// TwinCAT 3 PLC project RS485HausBus
// ProgramVersion: 3.1.4024.0
// libraries:
//   Tc2_SerialCom, * (Beckhoff Automation GmbH)
//   Tc2_Standard, * (Beckhoff Automation GmbH)
//   Tc2_System, * (Beckhoff Automation GmbH)
//   Tc3_Module, * (Beckhoff Automation GmbH)
// project tree:
//   DUTs/BusTaster/ ST_BusTaster6F_Cnt.TcDUT, ST_BusTaster6F_Input.TcDUT (not stored), ST_BusTaster6F_Output.TcDUT (not stored)
//   DUTs/RelaisModul/ ST_BusRelais16F_Cnt.TcDUT (not stored), ST_BusRelais16F_Input.TcDUT (not stored), ST_BusRelais16F_Output.TcDUT (not stored)
//   DUTs/Service/ ST_FiFoMaster_State.TcDUT (not stored), ST_RS485Startup_State.TcDUT
//   / GlobalTextList.TcGTLO, PlcTask.TcTTO, Visualisierungsmanager.TcVMO (not stored)
//   GVLs/ GVL.TcGVL, GVL_Constant.TcGVL, GVL_HausBus_Parameter.TcGVL (not stored), GVL_RS485FiFoSend.TcGVL, GVL_ServiceVisu.TcGVL
//   POUs/ RS485_COM_PRG.TcPOU
//   POUs/RS485_Hausbus_FB/BusTaster/ fb_StringConvTB6F.TcPOU, fb_TasterBus6F.TcPOU
//   POUs/RS485_Hausbus_FB/Events/ fb_BusBrsEvent.TcPOU, fb_BusPingEvent.TcPOU, fb_BusRhdEvent.TcPOU, fb_BusTasterEvent.TcPOU, fb_BusTempEvent.TcPOU
//   POUs/RS485_Hausbus_FB/RelaisModul/ fb_RelaisBus16F.TcPOU, fb_StringConvRB16F.TcPOU
//   POUs/RS485_Hausbus_FB/RS485 COM/FB/ fb_FilterArray.TcPOU
//   POUs/RS485_Hausbus_FB/RS485 COM/ fb_RS485ComCheck.TcPOU
//   POUs/RS485_Hausbus_FB/RS485 COM/RS485_Master/ fb_RS485FiFoMaster.TcPOU, fb_RS485Startup.TcPOU
//   VISUs/HausBus_RS485/ BusRelais16F_Frame.TcVIS, BusRS485Master_Frame.TcVIS, BusTatster6F_Frame.TcVIS, RS485HB_ServiceVISU.TcVIS

CONFIGURATION RS485HausBus
    RESOURCE PLC ON TwinCAT3
        TASK PlcTask(INTERVAL := T#1ms, PRIORITY := 20);
        PROGRAM RS485_COM_PRG WITH PlcTask : RS485_COM_PRG;
    END_RESOURCE
END_CONFIGURATION

// ---- DUTs/BusTaster/ST_BusTaster6F_Cnt.TcDUT
TYPE ST_BusTaster6F_Cnt :
STRUCT
	dwCntButtons    :ARRAY[1..6] OF DWORD;
END_STRUCT
END_TYPE

// ---- DUTs/Service/ST_RS485Startup_State.TcDUT
TYPE ST_RS485Startup_State :
STRUCT
	bBusOk					:BOOL;
	bStartupError			:BOOL;
	sStartupState			:STRING;
	bStartupDone			:BOOL;
END_STRUCT
END_TYPE

// ---- GVLs/GVL.TcGVL
{attribute 'Tc2GvlVarNames'}
VAR_GLOBAL

    KL6041In    					AT %I* : KL6inData22B; // Eingangsdaten von der Klemme
    KL6041Out 						AT %Q* : KL6outData22B; // Ausgangsdaten zur Klemme
	
	uiEtherCATStateBK1120_RS485COM	AT %I* : UINT;			// EtherCAT Status 
	uiKBusStateBK1120_RS485COM		AT %I* : UINT;			// Buskoppler Status
	
END_VAR

// ---- GVLs/GVL_Constant.TcGVL
{attribute 'Tc2GvlVarNames'}
VAR_GLOBAL CONSTANT
	cMaxBusTaster	:INT :=10;			// Anzahl der Bus Taster 
	cMaxBusRelais	:INT :=1;			// Anzahl der Bus Relais 
	cMaxRS485CMDFiFo	:INT := 15;		// Anzahl der Zeilen im FiFo Buffer (Achtung jder Bus Teilnehmer Benötigt eine Zeile! also immer cMaxBusTaster +cMaxBusRelais +etc.)  
END_VAR

// ---- GVLs/GVL_RS485FiFoSend.TcGVL
{attribute 'qualified_only'}
VAR_GLOBAL
	bSendDoneFiFo	:ARRAY[1..cMaxRS485CMDFiFo] OF BOOL;			(* Rückmeldung Aus dem FiFo Master Baustein, dass der Sendevorgang abgeschlossen ist *)
	sSendFiFo		:ARRAY[1..cMaxRS485CMDFiFo] OF STRING(255);		(* Zeile für den FiFo Master Baustein, von jedem einzelnen Busteilnehmer *)
END_VAR

// ---- GVLs/GVL_ServiceVisu.TcGVL
{attribute 'qualified_only'}
VAR_GLOBAL
	iDeviceTasterVisu			:INT := 1;
	iDeviceRelaisVisu			:INT := cMaxBusTaster+1;
	
	bTasterServiceAktiv			:ARRAY[1..cMaxBusTaster] OF BOOL;
	bRelaisServiceAktiv			:ARRAY[cMaxBusTaster+1..cMaxBusTaster+cMaxBusRelais+1] OF BOOL;
	stTasterService				:ARRAY[1..cMaxBusTaster] OF ST_BusTaster6F_Input;
	stRelaisService				:ARRAY[cMaxBusTaster+1..cMaxBusTaster+cMaxBusRelais+1] OF ST_BusRelais16F_Input;
	
END_VAR

// ---- POUs/RS485_COM_PRG.TcPOU
(*======================================================================================================================================*)
(*RS485_COM_PRG: Beispielhaftes Programm zum Steuern von HAus-Bus.de Komponenten über RS485 mit TwinCAT
					Achtung dieser POU muss als 1ms Task Aufgerufen werden um Ordnungsgemäß zu laufen *)
(*
Date          	| Version    	| created under        	| Author          	| Remark *)
(*====================================================================================================================================================*)
(*15/05/2025   	| 1.00      		| TC3		  		| N.Kersting       | first release *)
(*====================================================================================================================================================*)

PROGRAM RS485_COM_PRG
VAR  
    fbTaster 					:ARRAY[1..cMaxBusTaster] OF fb_TasterBus6F;	
	fbRelais					:ARRAY[cMaxBusTaster+1..cMaxBusRelais+cMaxBusTaster+1] OF fb_RelaisBus16F;
    i,h,j						:INT;
	
	fbRS485Startup				:fb_RS485Startup;		(* Startup Parametrierung der Klemme/ RS485 Bus *)
	fbRS485SendCmdFiFo			:fb_RS485FiFoMaster;	(* Sende und Empfangs FiFo für RS485 *)
	fbLineControl 				:SerialLineControl;		(* Hält die Serielle Kommunikation Aufrecht *)
	
	fComBufferReset				:ClearComBuffer;		(* Löschen des SPS Internen Bufferinhalts *)
	
	rxBuffer 					:ComBuffer;				(* COM Buffer Empfangen *)
    txBuffer 					:ComBuffer;				(* COM Buffer Senden *)
	
	
	
END_VAR

(* IDs Setzen *)
ac00_HausBusIdRS485COM();
(* RS485 Klemmen Config *)
ac01_StartupRS485COM();

ACTION ac00_HausBusIdRS485COM:
(* Initialisierung der Gerätenamen *)
(* Achtung nur Beispiele *)
fbTaster[1].I_stInput.sName := 		'Wohnzimmer';		(* Name, wie der Teilnehmer heißt / Bezeichnung *)
fbTaster[1].I_stInput.diID := 		5256;				(* Haus-Bus ID, welche auf dem Aufkleber steht  *)
		
fbTaster[2].I_stInput.sName := 		'Test1';
fbTaster[2].I_stInput.diID := 		5269;

fbTaster[3].I_stInput.sName := 		'Test2';
fbTaster[3].I_stInput.diID := 		2222;

fbTaster[4].I_stInput.sName := 		'Test3';
fbTaster[4].I_stInput.diID := 		3333;

fbTaster[5].I_stInput.sName := 		'Test4';
fbTaster[5].I_stInput.diID := 		4444;

fbTaster[6].I_stInput.sName := 		'Test5';
fbTaster[6].I_stInput.diID := 		5555;

fbTaster[7].I_stInput.sName := 		'Test6';
fbTaster[7].I_stInput.diID := 		6666;

fbTaster[8].I_stInput.sName := 		'Test7';
fbTaster[8].I_stInput.diID := 		7777;

fbTaster[9].I_stInput.sName := 		'Test8';
fbTaster[9].I_stInput.diID := 		8888;

fbTaster[10].I_stInput.sName := 	'Test9';
fbTaster[10].I_stInput.diID := 		9999;

fbRelais[11].I_stInput.sName := 	'Jalousie 1';
fbRelais[11].I_stInput.diID :=		5614;
END_ACTION

ACTION ac01_StartupRS485COM:

(* Klemmen Startup, inkl Klemmenkonfiguration usw. *)
fbRS485Startup(
	I_bExecute:= 		TRUE, 
	I_bBusOK:= 			uiEtherCATStateBK1120_RS485COM = 8
						AND uiKBusStateBK1120_RS485COM = 0, 
	I_tStartupVerz:= 	T#5S, 
	IQ_InData:= 		KL6041In, 
	IQ_OutData:= 		KL6041Out, 
	Q_sState=> , 
	Q_bStartupDone=> , 
	Q_bError=> );

(* Aktivierung der Linecontrole erst wenn Startup erfolgt *)	
IF fbRS485Startup.Q_bStartupDone
THEN
	fbLineControl(
		Mode := 		ComSerialLineMode_t.SERIALLINEMODE_KL6_22B_STANDARD,
		pComIn := 		ADR(KL6041In),
		pComOut := 		ADR(KL6041Out),
		SizeComIn := 	UINT_TO_INT(SIZEOF(KL6041In)),
		RxBuffer := 	rxBuffer,
		TxBuffer := 	txBuffer );
				
	(* Relais *)
	ac10_HausBusRelaisRS485COM();
	(* Taster *)
	ac10_HausBusTasterRS485COM();
	
	(* Senden FiFo *)
	fbRS485SendCmdFiFo(
		I_sSendCmdFiFo:= 		GVL_RS485FiFoSend.sSendFiFo, 
		I_bExecute:= 			TRUE, 
		I_bBusBelastungstest := ,
		I_bReset:= , 
		I_pTxBuffer:= 			ADR(txBuffer), 
		I_pRxBuffer:= 			ADR(rxBuffer), 
		Q_lrBusAuslastung=>		,
		Q_bBusy=> , 
		Q_bDone=> , 
		Q_bError=> , 
		Q_sState=> );
	
ELSE
	(* Com Buffer zum Resetten *)
	fComBufferReset(Buffer:= rxBuffer);
	fComBufferReset(Buffer:= txBuffer);
END_IF
END_ACTION

ACTION ac10_HausBusRelaisRS485COM:
(* BusRelais Aufrufe *)
FOR h := cMaxBusTaster +1 TO cMaxBusRelais+cMaxBusTaster+1 BY 1 DO (*cMaxBusTaster+1..cMaxBusRelais+cMaxBusTaster+1*)
		
	IF GVL_ServiceVisu.bRelaisServiceAktiv[h]
	THEN
		fbRelais[h].I_stInput.bOut := GVL_ServiceVisu.stRelaisService[h].bOut;
		fbRelais[h].I_stInput.bReset := GVL_ServiceVisu.stRelaisService[h].bReset;
	END_IF
	
	GVL_ServiceVisu.stRelaisService[h].sName :=	fbRelais[h].I_stInput.sName;
	GVL_ServiceVisu.stRelaisService[h].diID :=	fbRelais[h].I_stInput.diID;
	
	fbRelais[h].I_stInput.bExecute := TRUE;
	fbRelais[h](
		I_FifoID :=			h,
		I_bPingStart:= 		TRUE,	(* Direkt Starten *)
		I_StringReceived:=	fbRS485SendCmdFiFo.Q_sReceiveString);
		
	(* Sendebefehle an FiFo Übergeben *)
	GVL_RS485FiFoSend.sSendFiFo[h] :=	fbRelais[h].Q_sFiFoSend;	
END_FOR
END_ACTION

ACTION ac10_HausBusTasterRS485COM:
(* Bustaster Aufrufe *)
FOR i := 1 TO cMaxBusTaster BY 1 DO
			
	IF GVL_ServiceVisu.bTasterServiceAktiv[i]
	THEN
		fbTaster[i].I_stInput.iLED := GVL_ServiceVisu.stTasterService[i].iLED;
		fbTaster[i].I_stInput.iLEDBg := GVL_ServiceVisu.stTasterService[i].iLEDBg;
		fbTaster[i].I_stInput.iLEDExt := GVL_ServiceVisu.stTasterService[i].iLEDExt;
		fbTaster[i].I_stInput.bReset := GVL_ServiceVisu.stTasterService[i].bReset;
	END_IF
	
	GVL_ServiceVisu.stTasterService[i].sName :=	fbTaster[i].I_stInput.sName;
	GVL_ServiceVisu.stTasterService[i].diID :=	fbTaster[i].I_stInput.diID;
	
	fbTaster[i].I_stInput.bExecute := TRUE;
	fbTaster[i](
		I_FifoID :=			i,
		I_bPingStart:= 		TRUE , 	(* Taster Verzögert Pingen, damit weniger Busauslastung entsteht *)
		I_StringReceived:=	fbRS485SendCmdFiFo.Q_sReceiveString);
		
	(* Sendebefehle an FiFo Übergeben *)
	GVL_RS485FiFoSend.sSendFiFo[i] :=	fbTaster[i].Q_sFiFoSend;
END_FOR
END_ACTION

END_PROGRAM

// ---- POUs/RS485_Hausbus_FB/BusTaster/fb_TasterBus6F.TcPOU
(*======================================================================================================================================*)
(*FB_TasterBusSimple:	Einfache RS485 Kommunikation für Haus-bus.de Komponenten zum testen 	
						Achtung: Bei dem 6 Fach Taster ist zu Beachten, dass es nur 4 Externe EA/s gibt also 4 LEDs und 4 Taster *)
(*
Date          	| Version    	| created under        	| Author          	| Remark *)
(*====================================================================================================================================================*)
(*29/04/2025   	| 1.00      		| TC3		  		| N.Kersting       | first release *)
(*02/05/2025   	| 1.01      		| TC3		  		| N.Kersting       | Events für die Buttons werden erfolgreich verarbeitet *)
(*02/05/2025   	| 1.02      		| TC3		  		| N.Kersting       | Events für Temp, Helligkeit, Fuehctigkeit erfolgreich Implementier *)
(*02/05/2025   	| 1.03      		| TC3		  		| N.Kersting       | Set Schrittkette für Reset und LED Helligkeit erfolgreich Implementier*)
(*02/05/2025   	| 1.04      		| TC3		  		| N.Kersting       | In und Out Strukturen Implementiert und Startup nach Reset *)
(*02/05/2025   	| 1.05      		| TC3		  		| N.Kersting       | Pingabgfrage*)
(*02/05/2025   	| 1.06      		| TC3		  		| N.Kersting       | Reset Startup Implementiert*)
(*03/05/2025   	| 1.07      		| TC3		  		| N.Kersting       | Ping wird nun bei PLC Reset auch gestaret und Execute wird richtig verwendet*)
(*04/05/2025   	| 1.08      		| TC3		  		| N.Kersting       | Hintergrundbeleuchtung und Zähler für die Tatser Implementiert *)
(*04/05/2025   	| 1.09      		| TC3		  		| N.Kersting       | Neuen Baustein zum Einheitlichen versenden von Telegrammen Implementiert *)
(*05/05/2025   	| 2.00      		| TC3		  		| N.Kersting       | Komplett neuen Baustein, mit Externer Receive Auswertung und neuem Ping Baustein *)
(*06/05/2025   	| 2.01      		| TC3		  		| N.Kersting       | Externe LEDs Implementiert *)
(*07/05/2025   	| 2.02      		| TC3		  		| N.Kersting       | Im Startup wird nun auf die Device ID geachtet *)
(*08/05/2025   	| 2.03      		| TC3		  		| N.Kersting       | Externe LEDs sind nun Umschaltbar/ LEDs oder normaler Ausgang (Betriefft die Hintergrundbeleuchtung) -> Weniger Busauslastung *)
(*09/05/2025   	| 2.04      		| TC3		  		| N.Kersting       | Ping Versuche Implementiert mit Globalen Parametern *)
(*09/05/2025   	| 2.05      		| TC3		  		| N.Kersting       | Ping für Taster nun Auch automatisch durch Empfang von sämtlichen Telegrammen*)
(*09/05/2025   	| 2.06      		| TC3		  		| N.Kersting       | Bugfix im Startup Angepasst! nur noch Hintergrundbeleuchtung setzen! *)
(*10/05/2025   	| 3.00      		| TC3		  		| N.Kersting       | Umstellung auf Externe FiFo Sendebaustein *)
(*13/05/2025   	| 3.01      		| TC3		  		| N.Kersting       | Viele Bugs gefixt, bei Änderung der Ausgängen wird nun eine Anforderung gesetzt  *)
(*13/05/2025   	| 3.02      		| TC3		  		| N.Kersting       | Test für Github *)
(*====================================================================================================================================================*)
FUNCTION_BLOCK fb_TasterBus6F
VAR_INPUT
	I_FifoID			:INT;
	I_bPingStart		:BOOL;						(* Ping Done vom Vorheriegen*)
	I_stInput			:ST_BusTaster6F_Input;
	I_StringReceived	:STRING(255);
END_VAR
VAR_OUTPUT
	Q_sFiFoSend			:STRING(255);
   	Q_stOutput			:ST_BusTaster6F_Output;
	Q_stCnt				:ST_BusTaster6F_Cnt;
END_VAR
VAR
(*----------------------------------------------*)
(* Interne Parameter*)
(*----------------------------------------------*)		
	bSetExecute			:BOOL := TRUE;				(* Aktiviert die Schrittketten, welche Telegramme versenden *)
	bCheckPing			:BOOL := TRUE;				(* Ping Checken Schrittkette Aktivieren *)
	sStartZeichen		:BYTE := 16#FD;				(* Startzeichen Präfix *)
	sEndZeichen			:BYTE := 16#FE;				(* Endzeichen Suffix *)
	iAnzResetSend		:INT := 2;					(* Anzahl der Sendeversuche bei Reset *)
	tPingTimer			:TIME:= T#5S;				(* Zeit, bis wiederholend der Ping versendet wird *)
	tReceiveTimeout		:TIME:= T#2S;				(* Zeit, bis die Event Schrittkette für das Empfangen Automatisch neu Startet*)
	tStartupLEDOn		:TIME:= T#4S;				(* Zeit, wie Lange die LEDS beim Startup kurz eingeschaltet werden *)
	tResetTimeout		:TIME:= T#8S;				(* Zeit, bis bei einem Reset es zu einem Fehler kommt, wenn kein Ping empfangen wird *)
	tResetReboot		:TIME:= T#10S;				(* Zeit, die nach einem Reset Abgewaretet wird damit das Gerät neustarten kann*)
	tResetStartup		:TIME:= T#5S;				(* Zeit, die nach einem Reset Abgewaretet wird bis ein Startup ausgeführt wird nach dem erhalt des Pings vom Gerät*)
	tStartupAfterReset	:TIME := T#5S;				(* Zeit, wann das Startup Zurückgesetzt wird, wenn der Ping verloren wird *)
(*----------------------------------------------*)
(* Strings *)
(*----------------------------------------------*)			
	sSendString			:STRING(255);
	sFiFoSend			:STRING(255);
	sReceived			:STRING(255);
	sLastSendString		:STRING(255);
	sStateReset			:STRING;
(*----------------------------------------------*)
(* Funktionsbausteine *)
(*----------------------------------------------*)
	fbBusTasterEvent	:ARRAY[1..6] OF fb_BusTasterEvent;		(* Interne 6 Taster Abfragen *)
	fbBusTasterEventExt	:ARRAY[1..6] OF fb_BusTasterEvent;		(* Externe 6 Eingänge Abfragen *)
	fbBusTempEvent		:fb_BusTempEvent;
	fbBusBrsEvent		:fb_BusBrsEvent;
	fbBusRhdEvent		:fb_BusRhdEvent;
	fbStringConvTB6F	:fb_StringConvTB6F;
	fbRS485ComCheck		:fb_RS485ComCheck;
(*----------------------------------------------*)
(* Indexe *)
(*----------------------------------------------*)	
	iDeviceStartup		:INT :=0;	(* Startup Schrittkette *)
	sDeviceStartup		:STRING;
    iState     			:INT := 0;
	iStepSet			:INT;
	i,h,j,l,e			:INT;
	idxLED				:INT;
	idxBtn				:INT := 1;
	
	iDimmMem			:ARRAY[1..6] OF INT;
	iDimmMemExt			:ARRAY[1..6] OF INT;
	iDimmBGAnf			:INT;
	iDimmAnf			:ARRAY[1..6] OF INT;
	iDimmAnfExt			:ARRAY[1..6] OF INT;
	
	iDimmBgMem			:INT;
	cntChangesDimm		:INT;
	cntChangesDimmExt	:INT;
	icntResetSend		:INT;
	iMaxPingTry			:INT := 5;
(*----------------------------------------------*)
(* Timer/Trigger *)
(*----------------------------------------------*)		
	r_trigStartupAfterReset	:r_trig;
	r_TrigReset				:r_trig;		
	r_TrigCountBtn			:ARRAY[1..6] OF r_trig;
	
	tonStartupAfterReset	:ton;
	tonReceiveTimeout		:ton;
	tonResetTimeout			:ton;
	tonResetDone			:ton;
	tonStepStartup			:ton;
(*----------------------------------------------*)
(* Status *)
(*----------------------------------------------*)			
	bPingOK					:BOOL;
	bErrorEvent				:BOOL;
	bErrorPing				:BOOL;
	bErrorSet				:BOOL;
	bErrorReset				:BOOL;
	bResetBusy				:BOOL;
	bResetDone				:BOOL;
	bResetAutoStart			:BOOL;
	bStartupStart			:BOOL;
	bStartupDone			:BOOL;	
	bMemExt					:BOOL;
	bStartUpCheckPing		:BOOL;
	bActivateSend			:BOOL;
	bReadyToPing			:BOOL;
	bSendeAnforderung		:BOOL;
	bSendeAnforderungExt	:BOOL;
	bSendeAnforderungBG		:BOOL;
	
END_VAR

(*============================================================================================*)
(* Parameter *)
tPingTimer :=		GVL_HausBus_Parameter.cTimePingTimeTaster;
tReceiveTimeout :=	GVL_HausBus_Parameter.cTimeReceiveTimeoutTaster;
bCheckPing :=		GVL_HausBus_Parameter.bUseTasterPing;
iMaxPingTry :=		GVL_HausBus_Parameter.cMaxPingTry;

(*============================================================================================*)
(* Startup Zurücksetzen Reset *)
r_TrigReset(CLK := I_stInput.bReset);

(* Startup Zurücksetzen bei Busverlust *)
tonStartupAfterReset(
	IN := NOT bPingOK
			AND bCheckPing,
	PT:= tStartupAfterReset);

r_trigStartupAfterReset
	(CLK := tonStartupAfterReset.Q);
	
IF NOT I_stInput.bExecute
	OR r_TrigReset.Q
	OR r_trigStartupAfterReset.Q
THEN
	iDeviceStartup := 0;
END_IF

(*============================================================================================*)
(* Ping Dauerhaft Senden*)
ac02_Ping();
	
(*============================================================================================*)
(* Startup Schrittkette *)
CASE iDeviceStartup OF
(*============================================================================================*)
0: 	sDeviceStartup := 'INIT';
	bResetDone := FALSE;
	bStartupDone := FALSE;
	bStartupStart := FALSE;
	bResetAutoStart := FALSE;
	bStartUpCheckPing := FALSE;
	bActivateSend := FALSE;
	bReadyToPing := TRUE;
	sFiFoSend := ''; 
	iStepSet := 0;
	
	IF 	I_stInput.bExecute
	THEN
		iDeviceStartup := iDeviceStartup+1;
	END_IF
(*============================================================================================*)
1: 	sDeviceStartup := 'Device ID Prüfen';
	
	IF  I_stInput.diID <> 0
	THEN
		iDeviceStartup := iDeviceStartup+1;
	ELSE
		sDeviceStartup := 'ERROR- Device ID Prüfen';
	END_IF
(*============================================================================================*)
2: 	sDeviceStartup := 'Verbindung Prüfen';
	bStartUpCheckPing := TRUE;
	bActivateSend := TRUE;	(* Senden Aktivieren *)
	
	sDeviceStartup := CONCAT(sDeviceStartup,fbRS485ComCheck.Q_sState);
	
	IF fbRS485ComCheck.Q_bComOk
		OR NOT bCheckPing
	THEN
		iDeviceStartup := iDeviceStartup+1;
	END_IF

(*============================================================================================*)
3: 	sDeviceStartup := 'Reset Ausführen';	
	bActivateSend := TRUE;	(* Senden Aktivieren *)
	
	(*	RESET Device *)
	ac01_SetReset();
	bResetAutoStart := TRUE;
	
	sDeviceStartup :=	CONCAT(sDeviceStartup,sStateReset);
	
	IF bResetDone
	THEN
		iStepSet := 0;
		iDeviceStartup := iDeviceStartup+1;
	END_IF

(*============================================================================================*)
4: 	sDeviceStartup := 'Startup Ausführen';
		
	(* LED Setzen *)
	ac01_SetLED();
	
	bStartupStart := TRUE;
	
	IF bStartupDone 
	THEN
		bStartupStart := FALSE;
		iDeviceStartup := 999;
	END_IF

(*============================================================================================*)
999: 
	(*bReadyToPing := NOT fbRS485SendCmd.Q_bBusy;*)
	
	(* LED Setzen *)
	ac01_SetLED();
	
	(* Events Auslesen *)
	ac00_Event();
	
	(* Zähler *)
	ac10_Counter();
	
	sDeviceStartup := 'Startup Ausgeführt- Gerät im OP';
	
END_CASE

(*============================================================================================*)
(* Sendebaustein *)
IF bActivateSend
THEN
	IF fbRS485ComCheck.Q_sSend <>''
	THEN
		Q_sFiFoSend :=	fbRS485ComCheck.Q_sSend;
	ELSE
		Q_sFiFoSend :=	sFiFoSend;
	END_IF
END_IF

(*============================================================================================*)	
(* Zähler *)
ac10_Counter();
	
(*============================================================================================*)
(* Outputs *)
Q_stOutput.bCOM :=		bPingOK;

Q_stOutput.bError := 	bErrorEvent
						OR bErrorPing
						OR bErrorSet
						OR (NOT bPingOK
						AND bCheckPing);
						
Q_stOutput.bStartupDone	:=	bStartupDone;

Q_stOutput.sState :=	CONCAT(I_stInput.sName,'| ');
Q_stOutput.sState :=	CONCAT(Q_stOutput.sState, sDeviceStartup);

ACTION ac00_Event:
(*============================================================================================*)
(*	EVENT Schrittkette *)
(*============================================================================================*)
sReceived := I_StringReceived;
	
FOR i := 1 TO 6 BY 1 DO 
	fbBusTasterEvent[i](
		I_sID:= 				DINT_TO_STRING(I_stInput.diID), 
		I_sInstID:= 			INT_TO_STRING(i+16), 
		I_sReceivedString:= 	sReceived, 
		Q_bOut=> 				Q_stOutput.bButtons[i]);
	
	fbBusTasterEventExt[i](
		I_sID:= 				DINT_TO_STRING(I_stInput.diID), 
		I_sInstID:= 			INT_TO_STRING(i+32), 
		I_sReceivedString:= 	sReceived, 
		Q_bOut=> 				Q_stOutput.bButtonsExt[i]);
		
	fbBusTempEvent(
		I_sID:= 				DINT_TO_STRING(I_stInput.diID), 
		I_sInstID:= 			'1', 
		I_sReceivedString:= 	sReceived, 
		Q_lrTemp=> 				Q_stOutput.lrTemp);
		
	fbBusBrsEvent(
		I_sID:= 				DINT_TO_STRING(I_stInput.diID), 
		I_sInstID:= 			'1', 
		I_sReceivedString:= 	sReceived, 
		Q_lrBrs=> 				Q_stOutput.lrBrs);
		
	fbBusRhdEvent(
		I_sID:= 				DINT_TO_STRING(I_stInput.diID), 
		I_sInstID:= 			'1', 
		I_sReceivedString:= 	sReceived, 
		Q_lrRhd=> 				Q_stOutput.lrRhd);
END_FOR
END_ACTION

ACTION ac01_SetLED:
(*============================================================================================*)
(*	LED Helligkeit Setzen/ Startup Schrittkette *)
(*============================================================================================*)

(* Einfaches Setzen der LED Helligkeiten (0-100 Prozent *)
(* Neu, es werden alle LEDs zu einem String zusammengefügt und Gleichzeitig gesetzt *)
tonStepStartup(
	PT:= tStartupLEDOn);
	
cntchangesDimm := 0;
cntChangesDimmExt :=0;
	
FOR l := 1 TO 6 BY 1 DO
	IF iDimmMem[l] <> I_stInput.iLED[l]
	THEN
		cntChangesDimm := cntChangesDimm +1;
	END_IF

	IF  iDimmMemExt[l]<> I_stInput.iLEDExt[l]
	THEN
		cntChangesDimmExt := cntChangesDimmExt +1;
	END_IF
END_FOR

CASE iStepSet OF
(*============================================================================================*)
0:	(* INIT und warten auf Change *)				
	tonStepStartup.IN := FALSE;
	sFiFoSend := ''; 
	
	(* Änderungs- Anforderungen Prüfen*)
	FOR e := 1 TO 6 BY 1 DO
		IF cntChangesDimm<>0
		THEN
			(* Helligkeitanforderung Interne LEDs speichern *)
			bSendeAnforderung := TRUE;
			iDimmAnf[e] 	:= I_stInput.iLED[e];
		END_IF
		
		IF cntChangesDimmExt <> 0
		THEN
			(* Helligkeitanforderung Externe LEDs speichern *)
			bSendeAnforderungExt := TRUE;
			iDimmAnfExt[e] 	:= I_stInput.iLEDExt[e];
		END_IF
		
		IF I_stInput.iLEDBg <>iDimmBgMem
		THEN
			(* Helligkeitsanforderung Hintergrundbeleuchtung *)
			bSendeAnforderungBG := TRUE;
			iDimmBGAnf		:= I_stInput.iLEDBg;
		END_IF
	END_FOR
	
	(* Reagieren auf Anforderungen *)
	IF ((bSendeAnforderung
		OR bSendeAnforderungExt
		OR bSendeAnforderungBG)
		AND bSetExecute)
		AND fbRS485ComCheck.Q_sSend =''
		AND NOT bStartupStart
	THEN
		(* Helligkeitsvorgaben speichern in Mem Arrays *)
		FOR h := 1 TO 6 BY 1 DO
			iDimmMem[h] := I_stInput.iLED[h];
			iDimmMemExt[h] := I_stInput.iLEDExt[h];
			iDimmBgMem := I_stInput.iLEDBg;
		END_FOR
		
		iStepSet := 10;
	ELSIF
		bStartupStart
	THEN
		iStepSet := 100;	(* Startup *)
	END_IF
	
(*============================================================================================*)
10:	(* Prüfen welche Anforderung ausgeführt werden soll *)	
	IF	bSendeAnforderungBG
		AND NOT bSendeAnforderung
		AND NOT bSendeAnforderungExt 
	THEN
		iStepSet := 22;(* Direkt nur die Hintergrund Helligkeit setzen *)
	ELSE
		(* Nur Interne LEDs Schreiben *)
		IF bSendeAnforderung
			AND NOT bSendeAnforderungExt
			AND NOT bSendeAnforderungBG
		THEN
			fbStringConvTB6F(
				I_bSetBackground :=	FALSE,
				I_bReset :=			FALSE,
				I_bExtLED :=		FALSE,
				I_bHasExtLED :=		I_stInput.bExtOutLED,
				I_diID:= 			I_stInput.diID, 
				I_iLED:= 			iDimmAnf, 
				I_iLEDExt:=			iDimmAnfExt,
				I_iLEDBg:= 			iDimmBGAnf,		 
				I_sStartZeichen:= 	sStartZeichen, 
				I_sEndZeichen:= 	sEndZeichen, 
				Q_sConvString=> 	sSendString);
				
			(* Senden an FiFo*)
			IF GVL_RS485FiFoSend.bSendDoneFiFo[I_FifoID]
			THEN
				sFiFoSend :=	sSendString;
			END_IF
			IF NOT GVL_RS485FiFoSend.bSendDoneFiFo[I_FifoID]
			THEN
				bSendeAnforderung := FALSE;
				sLastSendString :=	sFiFoSend;
				iStepSet := 20;
			END_IF
		ELSIF
			(* Nur Externe LEDs Schreiben *)	
			bSendeAnforderungExt
			AND NOT bSendeAnforderung
			AND NOT bSendeAnforderungBG
		THEN
			fbStringConvTB6F(
				I_bSetBackground :=	FALSE,
				I_bReset :=			FALSE,
				I_bExtLED :=		TRUE,
				I_bHasExtLED :=		I_stInput.bExtOutLED,
				I_diID:= 			I_stInput.diID, 
				I_iLED:= 			iDimmAnf, 
				I_iLEDExt:=			iDimmAnfExt,
				I_iLEDBg:= 			iDimmBGAnf,				 
				I_sStartZeichen:= 	sStartZeichen, 
				I_sEndZeichen:= 	sEndZeichen, 
				Q_sConvString=> 	sSendString);
			
			(* Senden an FiFo*)
			IF GVL_RS485FiFoSend.bSendDoneFiFo[I_FifoID]
			THEN
				sFiFoSend :=	sSendString;
			END_IF
			IF NOT GVL_RS485FiFoSend.bSendDoneFiFo[I_FifoID]
			THEN
				bSendeAnforderungExt := FALSE;
				sLastSendString :=	sFiFoSend;
				iStepSet := 20;
			END_IF
		ELSE
			(* Externe und Interne LEDs Schreiben *)
			bMemExt := TRUE; (* Speichern, damit anschließend noch die Externen LEDs gesetzt werden *)
			
			fbStringConvTB6F(
				I_bSetBackground :=	FALSE,
				I_bReset :=			FALSE,
				I_bExtLED :=		FALSE,
				I_bHasExtLED :=		I_stInput.bExtOutLED,
				I_diID:= 			I_stInput.diID, 
				I_iLED:= 			iDimmAnf, 
				I_iLEDExt:=			iDimmAnfExt,
				I_iLEDBg:= 			iDimmBGAnf,			 
				I_sStartZeichen:= 	sStartZeichen, 
				I_sEndZeichen:= 	sEndZeichen, 
				Q_sConvString=> 	sSendString);
			
			(* Senden an FiFo*)
			IF GVL_RS485FiFoSend.bSendDoneFiFo[I_FifoID]
			THEN
				sFiFoSend :=	sSendString;
			END_IF
			IF NOT GVL_RS485FiFoSend.bSendDoneFiFo[I_FifoID]
			THEN
				bSendeAnforderung := FALSE;
				bSendeAnforderungExt := FALSE;
				sLastSendString :=	sFiFoSend;
				iStepSet := 20;
			END_IF
		END_IF
	END_IF
(*============================================================================================*)	
20:	(* Warten bis nicht Busy *)	
	
	IF GVL_RS485FiFoSend.bSendDoneFiFo[I_FifoID]
	THEN
		sFiFoSend := ''; 
		IF NOT bMemExt
		THEN
			IF bSendeAnforderungBG
			THEN
				iStepSet := 22;
			ELSE
				iStepSet := 0;
			END_IF
		ELSE
			iStepSet :=	21;
		END_IF
	END_IF
	
(*============================================================================================*)	
21:	(* Externe LEDs Senden *)	
	bMemExt := FALSE;
	bSendeAnforderungExt := FALSE;
	
	fbStringConvTB6F(
		I_bSetBackground :=	FALSE,
		I_bReset :=			FALSE,
		I_bExtLED :=		TRUE,
		I_bHasExtLED :=		I_stInput.bExtOutLED,
		I_diID:= 			I_stInput.diID, 
		I_iLED:= 			iDimmAnf, 
		I_iLEDExt:=			iDimmAnfExt,
		I_iLEDBg:= 			iDimmBGAnf,				 
		I_sStartZeichen:= 	sStartZeichen, 
		I_sEndZeichen:= 	sEndZeichen, 
		Q_sConvString=> 	sSendString);
		
	(* Senden an FiFo*)
	IF GVL_RS485FiFoSend.bSendDoneFiFo[I_FifoID]
	THEN
		sFiFoSend :=	sSendString;
	END_IF
	IF NOT GVL_RS485FiFoSend.bSendDoneFiFo[I_FifoID]
	THEN
		sLastSendString :=	sFiFoSend;
		iStepSet := 20;
	END_IF
	
(*============================================================================================*)	
22:	(* Hintergrundbeleuchtung senden *)		
	bSendeAnforderungBG := FALSE;
	
	fbStringConvTB6F(
		I_bSetBackground :=	TRUE,
		I_bReset :=			FALSE,
		I_bExtLED :=		FALSE,
		I_bHasExtLED :=		I_stInput.bExtOutLED,
		I_diID:= 			I_stInput.diID, 
		I_iLED:= 			iDimmAnf, 
		I_iLEDExt:=			iDimmAnfExt,
		I_iLEDBg:= 			iDimmBGAnf,			 
		I_sStartZeichen:= 	sStartZeichen, 
		I_sEndZeichen:= 	sEndZeichen, 
		Q_sConvString=> 	sSendString);
		
	(* Senden an FiFo*)
	IF GVL_RS485FiFoSend.bSendDoneFiFo[I_FifoID]
	THEN
		sFiFoSend :=	sSendString;
	END_IF
	IF NOT GVL_RS485FiFoSend.bSendDoneFiFo[I_FifoID]
	THEN
		sLastSendString :=	sFiFoSend;
		iStepSet := 20;
	END_IF

(*============================================================================================*)	
(* Startup LEDS einmal Einschalten *)
100:	tonStepStartup.IN := TRUE;
	
	IF tonStepStartup.Q
	THEN
		iStepSet := 110;
	END_IF
	
(*============================================================================================*)
110:	(* String senden *)	
	tonStepStartup.IN := FALSE;
	
	fbStringConvTB6F(
		I_bSetBackground :=	TRUE,
		I_bExtLED :=		FALSE,
		I_bReset :=			FALSE,
		I_bHasExtLED :=		I_stInput.bExtOutLED,
		I_diID:= 			I_stInput.diID, 
		I_iLEDBg:= 			100,		 
		I_sStartZeichen:= 	sStartZeichen, 
		I_sEndZeichen:= 	sEndZeichen, 
		Q_sConvString=> 	sSendString);
			
	(* Senden an FiFo*)
	IF GVL_RS485FiFoSend.bSendDoneFiFo[I_FifoID]
	THEN
		sFiFoSend :=	sSendString;
	END_IF
	IF NOT GVL_RS485FiFoSend.bSendDoneFiFo[I_FifoID]
	THEN
		
		iStepSet := 111;
	END_IF
	
(*============================================================================================*)	
111:(* Warten bis nicht Busy *)	
	IF GVL_RS485FiFoSend.bSendDoneFiFo[I_FifoID]
	THEN
		sFiFoSend := ''; 
		tonStepStartup.IN := TRUE;
		
		IF tonStepStartup.Q
		THEN
			tonStepStartup.IN := FALSE;
			iStepSet := 120;
		END_IF
	END_IF
	
(*============================================================================================*)
120:	(* String senden *)	
	fbStringConvTB6F(
		I_bSetBackground :=	TRUE,
		I_bExtLED :=		FALSE,
		I_bReset :=			FALSE,
		I_bHasExtLED :=		I_stInput.bExtOutLED,
		I_diID:= 			I_stInput.diID, 
		I_iLEDBg:= 			0,		 
		I_sStartZeichen:= 	sStartZeichen, 
		I_sEndZeichen:= 	sEndZeichen, 
		Q_sConvString=> 	sSendString);
			
	(* Senden an FiFo*)
	IF GVL_RS485FiFoSend.bSendDoneFiFo[I_FifoID]
	THEN
		sFiFoSend :=	sSendString;
	END_IF
	IF NOT GVL_RS485FiFoSend.bSendDoneFiFo[I_FifoID]
	THEN
		iStepSet := 130;
	END_IF
	
(*============================================================================================*)	
130:(* Warten bis nicht Busy *)	
	IF GVL_RS485FiFoSend.bSendDoneFiFo[I_FifoID]
	THEN
		sFiFoSend := ''; 
			
		tonStepStartup.IN := TRUE;
	
		IF tonStepStartup.Q
		THEN
			bStartupDone := TRUE;
			tonStepStartup.IN := FALSE;
			bStartupStart := FALSE;
			iStepSet := 10;	(* Anschließend noch einmal die Eingangs Helligkeit setzen *)
		END_IF
	END_IF	

END_CASE

(*bErrorSet := fbRS485SendCmd.Q_bError;*)
END_ACTION

ACTION ac01_SetReset:
(*============================================================================================*)
(*	RESET Schrittkette *)
(*============================================================================================*)
tonResetTimeout(
	PT := tResetTimeout);

tonResetDone();

(* Einfaches Setzen der LED Helligkeiten (0-100 Prozent *)
CASE iStepSet OF
(*============================================================================================*)
0:	sStateReset := 'INIT';
	
	IF (bSetExecute
		AND (I_stInput.bReset
		OR bResetAutoStart))
	THEN
		sFiFoSend := ''; 
		bStartupDone := FALSE;
		bResetDone := FALSE;
		tonResetTimeout.IN := FALSE;
		tonResetDone.IN := FALSE;
		icntResetSend := 0;
		
		(* Ausgänge alle auf 0 setzen *)
		FOR h := 1 TO 6 BY 1 DO
			fbBusTasterEvent[i](
				I_sReceivedString :='');
				
			fbBusTasterEventExt[i](
				I_sReceivedString :='');	
				
			iDimmMem[h] := 0;
			Q_stOutput.bButtons[h] := FALSE;
			Q_stOutput.lrTemp := 0;
			Q_stOutput.lrBrs := 0;
			Q_stOutput.lrRhd := 0;
		END_FOR
		
		fbBusTempEvent(
			I_sReceivedString :='',	
			I_bReset := TRUE);
			
		fbBusBrsEvent(
			I_sReceivedString :='',	
			I_bReset := TRUE);
			
		fbBusRhdEvent(
			I_sReceivedString :='',	
			I_bReset := TRUE);
		
		bPingOK := FALSE;
		
		iStepSet := iStepSet +1;
	END_IF

(*============================================================================================*)	
1:	sStateReset := 'Sende Reset Befehl';
	bResetBusy := TRUE;
	bErrorReset := FALSE;
	
	fbStringConvTB6F(
		I_bReset :=			TRUE,
		I_diID:= 			I_stInput.diID, 		 
		I_sStartZeichen:= 	sStartZeichen, 
		I_sEndZeichen:= 	sEndZeichen, 
		Q_sConvString=> 	sSendString);

	(* Senden an FiFo*)
	IF GVL_RS485FiFoSend.bSendDoneFiFo[I_FifoID]
	THEN
		sFiFoSend :=	sSendString;
	END_IF
	IF NOT GVL_RS485FiFoSend.bSendDoneFiFo[I_FifoID]
	THEN
		iStepSet := iStepSet+1;
	END_IF

(*============================================================================================*)
2:	sStateReset := 'Sende Reset Befehl';

	IF GVL_RS485FiFoSend.bSendDoneFiFo[I_FifoID]
	THEN
		sFiFoSend := ''; 
		fbStringConvTB6F(
			I_bReset :=			FALSE);
		iStepSet := 3;
				
	END_IF
	
(*============================================================================================*)	
3:	sStateReset := 'Reset durchgeführt, Warte auf Ping';
	tonResetDone.IN := TRUE;
	tonResetDone.PT := tResetReboot;
	
	fbBusTempEvent(I_bReset := FALSE);
	fbBusBrsEvent(I_bReset := FALSE);
	fbBusRhdEvent(I_bReset := FALSE);
	
	iState := 0;
	
	IF tonResetDone.Q
	THEN
		tonResetDone.IN := FALSE;
		iStepSet := 4;
	END_IF
	
(*============================================================================================*)	
4:	sStateReset := 'Warte auf Ping vom Gerät';	
	tonResetTimeout.IN := TRUE;
	
	IF bPingOK 
		OR NOT bCheckPing
	THEN
		bErrorReset := FALSE;
		tonResetTimeout.IN := FALSE;
		iStepSet := 5;
	ELSIF
		tonResetTimeout.Q
	THEN
		sStateReset := 'Ping Timeout, keine Kommunikation';
		bErrorReset := TRUE;

		IF I_stInput.bReset
		THEN
			bResetBusy := FALSE;
			iStepSet := 0;
		END_IF
	END_IF

(*============================================================================================*)
5:	sStateReset := 'Startup Aktiv';
	
	tonResetDone.IN := NOT I_stInput.bReset;
	tonResetDone.PT := tResetStartup;
	sFiFoSend := ''; 
	
	IF tonResetDone.Q
	THEN
		fbStringConvTB6F(
			I_bReset :=			FALSE);
			
		sStateReset := 'Ping erhalten, Reset Erfolgreich';
		bResetAutoStart := FALSE;
		bResetDone := TRUE;
		bResetBusy := FALSE;
		iState := 0;
		iStepSet := 0;
	END_IF
END_CASE
END_ACTION

ACTION ac02_Ping:
(*============================================================================================*)
(* 	Ping Bautsein, Checkt ob die Kommunikation vorhanden ist *)
(*============================================================================================*)
fbRS485ComCheck(
	I_FifoID:=				I_FifoID,
	I_bExecute:= 			bCheckPing
							AND bStartUpCheckPing
							(*AND bReadyToPing*), 
	I_bStart :=				I_bPingStart,
	I_bTasterMode:=			TRUE,
	I_StringReceived:=		I_StringReceived,
	I_tPingIntervall:= 		tPingTimer, 
	I_tPingTimeout:= 		tReceiveTimeout, 
	I_diID:= 				I_stInput.diID, 
	I_sPingSymbol:= 		'.BTN.', 
	I_iInstID:= 			17, 
	I_sStartZeichen:= 		sStartZeichen, 
	I_sEndZeichen:= 		sEndZeichen, 
	I_iMaxPingTry :=		iMaxPingTry,	 
	Q_bComOk=> 				bPingOK, 
	Q_bError=> 				bErrorPing,
	Q_bSendDone=>			(* *));
END_ACTION

ACTION ac10_Counter:
(*============================================================================================*)
(* 	Zähler *)
(*============================================================================================*)
FOR j := 1 TO 6 BY 1 DO 
	r_TrigCountBtn[j](
		CLK := Q_stOutput.bButtons[j]);
		
	IF r_TrigCountBtn[j].Q
	THEN
		Q_stCnt.dwCntButtons[j] := Q_stCnt.dwCntButtons[j]+1;
	END_IF
	
END_FOR
END_ACTION

ACTION ac99_Doku:
(*======================================================================================================================================*)
(*	DOKU	*)
(*======================================================================================================================================*)
(* Wichtiger Hinweis:
		-Bei dem 6 Fach Taster ist zu Beachten, dass es nur 4 Externe EA/s gibt also 4 LEDs und 4 Taster, 
		da der ESP 32 Nur 10Es und 10As besitzt.
		- Die 4 Zusätzlichen Ausgänge werden von der Hintergrundbeleuchtung Ausgeschlossen und müssen über den Befehl: SET_MBR einzeln 
			gesetzt werden! *)	
	
(* Verdrahtung:		
	Verdrahtung füR: KL6041
        +-------+
        |       |
        | TxD+ ----+
        |         |----> RS485 A (zum Bus)
        | RxD+ ----+
        |         |
        | TxD− ----+
        |         |----> RS485 B (zum Bus)
        | RxD− ----+
        +-------+	*)
		
(*======================================================================================================================================*)
(* Telegrammbeschreibung *)

(*	Die XML Dateien der verschiedenen Module sind grundsätzlich immer gleich aufgebaut. 
	Je Instanz der verschiedenen Sensoren und Aktoren werden die zu sendenden Befehle bzw. 
	die zu empfangenen Events beschrieben. 
	Alle Telegramme sind ASCII kodiert und sind umgeben mit dem binären Startzeichen 0xFD und dem binären Endezeichen 0xFE.

	Grundaufbauer aller im Folgenden beschriebenen Telegramme:
	
	-Startzeichen immer 0xFD.
	-Punkte dienen als Trennzeichen der verschiedenen Elemente
	-Endezeichen immer 0xFE.
	-Element 1 ist die Geräte-ID, die entsprechend der verwendeten Module angepasst werden muss (hier beispielhaft jeweils 12345)
	-Element 2 ist ein Schlüsselwort für den jeweiligen Funktionstyp (z.b. BTN, LED, DIM, usw)
	-Element 3 ist die InstanzID gemäß XML Templates (also welche Taster oder welcher Dimmer konkret gemeint ist)
	-Element 4 zeigt die jeweilige Aktion zum Funktionstypen (z.b. ON, OFF, STATUS)
	-Anschließend kommen optional diverse Parameter, die mit P1,P2,...P3 bezeichnet werden
	
	Im Folgenden wird nur noch auf die speziellen Telegramdaten eingegangen:
	
	(*------------------------------------------------------------*)
	Taster oder digitaler Eingang (Sensor):
	(*------------------------------------------------------------*)
	Telegram Event:  	
	
	\xFD 12345.BTN.17.STATUS.P1 \xFE
	
		Funktionstyp:		BTN (kurz für Button)
		Instanz-ID:			hier 17 (in XML nachschauen)
		Aktion:				STATUS
		P1:					1, wenn Taste gedrückt bzw. Eingang aktiv
							0, wenn Taste losgelassen bzw. Eingang inaktiv
	
	Telegram Statusabfrage:  	
	
	\xFD 12345.BTN.17.gSTATUS \xFE
	
		Antwort:  			\xFD 12345.BTN.17.rSTATUS.P1 \xFE
		P1:					1, wenn Taste gedrückt bzw. Eingang aktiv
							0, wenn Taste losgelassen bzw. Eingang inaktiv

	(*------------------------------------------------------------*)
	Led (Aktor):
	(*------------------------------------------------------------*)
	Telegram Helligkeit setzen:  	
	
	\xFD 12345.LED.50.ON.P1.P2.P3 \xFE
	
		Funktionstyp:			LED
		Instanz-ID:				hier 50 (in XML nachschauen)
		Aktion:					ON
		P1:						gewünschte Helligkeit 0-100
		P2:						Einschaltdauer in 100stel Sekunden (0 = daueran)
		P3:						Einschaltverzögerung in Sekunden (0 = ohne Verzögerung)
	
	Telegram Mindesthelligkeit:  	
	
	\xFD 12345.LED.50.SET_MBR.P1 \xFE
		
		Aktion:					SET_MBR (Setzt eine Mindesthelligkeit, die auch dann erhalten bleibt, wenn man per OFF ausschaltet)
		P1:						gewünschte Helligkeit 0-100
	
	Telegram Statusabfrage:  	

	\xFD 12345.LED.50.gSTATUS \xFE
	
		Antwort:  				\xFD 12345.LED.50.rSTATUS.P1.P2 \xFE
		P1:						aktuelle Helligkeit 0-100
		P2:						Einschaltdauer in 100stel Sekunden
	
	(*------------------------------------------------------------*)
	Hintergrundbeleuchtung (Aktor):
	(*------------------------------------------------------------*)
	Telegram Minhelligkeit:  
	
	\xFD 12345.LBN.16.SET_MBR.P1 \xFE
	
		Aktion:					SET_MBR ((Setzt eine Mindesthelligkeit, die auch dann erhalten bleibt, wenn man per OFF ausschaltet)
		P1:						gewünschte Helligkeit 0-100
		
	Telegram Statusabfrage:  	

	\xFD 12345.LBN.16.gSTATUS \xFE
	
		Antwort:  				\xFD 12345.LBN.16.rSTATUS.P1 \xFE
		P1:						aktuelle Helligkeit 0-100

	(*------------------------------------------------------------*)
	Temperatursensor (Sensor):
	(*------------------------------------------------------------*)
	Telegram Event:  	
	
	\xFD 12345.TMP.1.STATUS.P1.P2 \xFE
	
		Funktionstyp:			TMP (kurz für Temperatur)
		Instanz-ID:				hier 1 (in XML nachschauen)
		Aktion:					STATUS
		P1:						Temperatur in Grad Vorkommastellen
		P2:						Temperatur in Grad Nachkommastellen
	
	Telegram Statusabfrage:  
	
	\xFD 12345.TMP.1.gSTATUS \xFE
	
		Antwort:  				\xFD 12345.TMP.1.rSTATUS.P1.P2 \xFE
		P1:						Temperatur in Grad Vorkommastellen
		P2:						Temperatur in Grad Nachkommastellen

	(*------------------------------------------------------------*)
	Feuchtesensor (Sensor):
	(*------------------------------------------------------------*)
	Telegram Event:  	

	\xFD 12345.RHD.1.STATUS.P1.P2 \xFE
	
		Funktionstyp:			RHD (kurz für Relative Humidity)
		Instanz-ID:				hier 1 (in XML nachschauen)
		Aktion:					STATUS
		P1:						Relative Luftfeuchtigkeit 0-100 Vorkommastellen
		P2:						Relative Luftfeuchtigkeit 0-100 Nachkommastellen

	Telegram Statusabfrage:  	
	
	\xFD 12345.RHD.1.gSTATUS \xFE
	
	Antwort:  					\xFD 12345.RHD.1.rSTATUS.P1 \xFE
	P1:							Relative Luftfeuchtigkeit 0-100 Vorkommastellen
	P2:							Relative Luftfeuchtigkeit 0-100 Nachkommastellen

	(*------------------------------------------------------------*)
	Helligkeitssensor (Sensor):
	(*------------------------------------------------------------*)
	Telegram Event:  	
	
	\xFD 12345.BRS.23.STATUS.P1.P2 \xFE
	
		Funktionstyp:			BRS (kurz für Brightness Sensor)
		Instanz-ID:				hier 23 (in XML nachschauen)
		Aktion:					STATUS
		P1:						Relative Helligkeit 0-255 Vorkommastellen
		P2:						Relative Helligkeit 0-255 Nachkommastellen
	
	Telegram Statusabfrage:  	
	
	\xFD 12345.BRS.23.gSTATUS \xFE
	
	Antwort:  					\xFD 12345.BRS.23.rSTATUS.P1 \xFE
	P1:							Relative Helligkeit 0-255 Vorkommastellen
	P2:							Relative Helligkeit 0-255 Nachkommastellen

(*======================================================================================================================================*)
(* Alle Telegramme im Überblick *)	

	<?xml version="1.0" encoding="utf-8"?>
	<Comm Title="Haus-Bus ID 12345" Comment="" Baudrate="57600" Databits="8" Parity="1" EndChar="510">
	<CommCmd Title="6-fach Taster 12345 - Hintergrundbeleuchtung" Comment="" CmdOn="\xFD12345.LBN.16.SET_MBR.&lt;v&gt;.0\xFE" CmdOff="\xFD12345.LBN.16.SET_MBR.0\xFE" Unit="" Analog="true" Text="false" Sensor="false" SourceValHigh="100" DestValHigh="100"/>
	<CommCmd Title="6-fach Taster 12345 - Temperatursensor" Comment="" CmdOn="\xFD12345.TMP.1.STATUS.\v\xFE" CmdOff="" Unit="&lt;v.2&gt;" Analog="true" Text="false" Sensor="true" SourceValHigh="100" DestValHigh="100"/>
	<CommCmd Title="6-fach Taster 12345 - Feuchtesensor" Comment="" CmdOn="\xFD12345.RHD.1.STATUS.\v\xFE" CmdOff="" Unit="&lt;v.x&gt;" Analog="true" Text="false" Sensor="true" SourceValHigh="100" DestValHigh="100"/>
	<CommCmd Title="6-fach Taster 12345 - Helligkeitssensor" Comment="" CmdOn="\xFD12345.BRS.1.STATUS.\v\xFE" CmdOff="" Unit="&lt;v.x&gt;" Analog="true" Text="false" Sensor="true" SourceValHigh="100" DestValHigh="100"/>
	<CommCmd Title="6-fach Taster 12345 - Led 1" Comment="" CmdOn="\xFD12345.LED.49.ON.&lt;v&gt;.0\xFE" CmdOff="\xFD12345.LED.49.OFF\xFE" Unit="" Analog="true" Text="false" Sensor="false" SourceValHigh="100" DestValHigh="100"/>
	<CommCmd Title="6-fach Taster 12345 - Led 2" Comment="" CmdOn="\xFD12345.LED.50.ON.&lt;v&gt;.0\xFE" CmdOff="\xFD12345.LED.50.OFF\xFE" Unit="" Analog="true" Text="false" Sensor="false" SourceValHigh="100" DestValHigh="100"/>
	<CommCmd Title="6-fach Taster 12345 - Led 3" Comment="" CmdOn="\xFD12345.LED.51.ON.&lt;v&gt;.0\xFE" CmdOff="\xFD12345.LED.51.OFF\xFE" Unit="" Analog="true" Text="false" Sensor="false" SourceValHigh="100" DestValHigh="100"/>
	<CommCmd Title="6-fach Taster 12345 - Led 4" Comment="" CmdOn="\xFD12345.LED.52.ON.&lt;v&gt;.0\xFE" CmdOff="\xFD12345.LED.52.OFF\xFE" Unit="" Analog="true" Text="false" Sensor="false" SourceValHigh="100" DestValHigh="100"/>
	<CommCmd Title="6-fach Taster 12345 - Led 5" Comment="" CmdOn="\xFD12345.LED.53.ON.&lt;v&gt;.0\xFE" CmdOff="\xFD12345.LED.53.OFF\xFE" Unit="" Analog="true" Text="false" Sensor="false" SourceValHigh="100" DestValHigh="100"/>
	<CommCmd Title="6-fach Taster 12345 - Led 6" Comment="" CmdOn="\xFD12345.LED.54.ON.&lt;v&gt;.0\xFE" CmdOff="\xFD12345.LED.54.OFF\xFE" Unit="" Analog="true" Text="false" Sensor="false" SourceValHigh="100" DestValHigh="100"/>
	<CommCmd Title="6-fach Taster 12345 - Taster 1" Comment="" CmdOn="\xFD12345.BTN.17.STATUS.\v\xFE" CmdOff="" Unit="&lt;v.x&gt;" Analog="true" Text="false" Sensor="true" SourceValHigh="100" DestValHigh="100"/>
	<CommCmd Title="6-fach Taster 12345 - Taster 2" Comment="" CmdOn="\xFD12345.BTN.18.STATUS.\v\xFE" CmdOff="" Unit="&lt;v.x&gt;" Analog="true" Text="false" Sensor="true" SourceValHigh="100" DestValHigh="100"/>
	<CommCmd Title="6-fach Taster 12345 - Taster 3" Comment="" CmdOn="\xFD12345.BTN.19.STATUS.\v\xFE" CmdOff="" Unit="&lt;v.x&gt;" Analog="true" Text="false" Sensor="true" SourceValHigh="100" DestValHigh="100"/>
	<CommCmd Title="6-fach Taster 12345 - Taster 4" Comment="" CmdOn="\xFD12345.BTN.20.STATUS.\v\xFE" CmdOff="" Unit="&lt;v.x&gt;" Analog="true" Text="false" Sensor="true" SourceValHigh="100" DestValHigh="100"/>
	<CommCmd Title="6-fach Taster 12345 - Taster 5" Comment="" CmdOn="\xFD12345.BTN.21.STATUS.\v\xFE" CmdOff="" Unit="&lt;v.x&gt;" Analog="true" Text="false" Sensor="true" SourceValHigh="100" DestValHigh="100"/>
	<CommCmd Title="6-fach Taster 12345 - Taster 6" Comment="" CmdOn="\xFD12345.BTN.22.STATUS.\v\xFE" CmdOff="" Unit="&lt;v.x&gt;" Analog="true" Text="false" Sensor="true" SourceValHigh="100" DestValHigh="100"/>
	<CommCmd Title="6-fach Taster 12345 - Extern Taster 1" Comment="" CmdOn="\xFD12345.BTN.33.STATUS.\v\xFE" CmdOff="" Unit="&lt;v.x&gt;" Analog="true" Text="false" Sensor="true" SourceValHigh="100" DestValHigh="100"/>
	<CommCmd Title="6-fach Taster 12345 - Extern Taster 2" Comment="" CmdOn="\xFD12345.BTN.34.STATUS.\v\xFE" CmdOff="" Unit="&lt;v.x&gt;" Analog="true" Text="false" Sensor="true" SourceValHigh="100" DestValHigh="100"/>
	<CommCmd Title="6-fach Taster 12345 - Extern Taster 3" Comment="" CmdOn="\xFD12345.BTN.35.STATUS.\v\xFE" CmdOff="" Unit="&lt;v.x&gt;" Analog="true" Text="false" Sensor="true" SourceValHigh="100" DestValHigh="100"/>
	<CommCmd Title="6-fach Taster 12345 - Extern Taster 4" Comment="" CmdOn="\xFD12345.BTN.36.STATUS.\v\xFE" CmdOff="" Unit="&lt;v.x&gt;" Analog="true" Text="false" Sensor="true" SourceValHigh="100" DestValHigh="100"/>
	<CommCmd Title="6-fach Taster 12345 - Extern Taster 5" Comment="" CmdOn="\xFD12345.BTN.37.STATUS.\v\xFE" CmdOff="" Unit="&lt;v.x&gt;" Analog="true" Text="false" Sensor="true" SourceValHigh="100" DestValHigh="100"/>
	<CommCmd Title="6-fach Taster 12345 - Extern Taster 6" Comment="" CmdOn="\xFD12345.BTN.38.STATUS.\v\xFE" CmdOff="" Unit="&lt;v.x&gt;" Analog="true" Text="false" Sensor="true" SourceValHigh="100" DestValHigh="100"/>
	<CommCmd Title="6-fach Taster 12345 - Extern Led 1" Comment="" CmdOn="\xFD12345.LED.65.ON.&lt;v&gt;.0\xFE" CmdOff="\xFD12345.LED.65.OFF\xFE" Unit="" Analog="true" Text="false" Sensor="false" SourceValHigh="100" DestValHigh="100"/>
	<CommCmd Title="6-fach Taster 12345 - Extern Led 2" Comment="" CmdOn="\xFD12345.LED.66.ON.&lt;v&gt;.0\xFE" CmdOff="\xFD12345.LED.66.OFF\xFE" Unit="" Analog="true" Text="false" Sensor="false" SourceValHigh="100" DestValHigh="100"/>
	<CommCmd Title="6-fach Taster 12345 - Extern Led 3" Comment="" CmdOn="\xFD12345.LED.67.ON.&lt;v&gt;.0\xFE" CmdOff="\xFD12345.LED.67.OFF\xFE" Unit="" Analog="true" Text="false" Sensor="false" SourceValHigh="100" DestValHigh="100"/>
	<CommCmd Title="6-fach Taster 12345 - Extern Led 4" Comment="" CmdOn="\xFD12345.LED.68.ON.&lt;v&gt;.0\xFE" CmdOff="\xFD12345.LED.68.OFF\xFE" Unit="" Analog="true" Text="false" Sensor="false" SourceValHigh="100" DestValHigh="100"/>
	<CommCmd Title="6-fach Taster 12345 - Extern Led 5" Comment="" CmdOn="\xFD12345.LED.69.ON.&lt;v&gt;.0\xFE" CmdOff="\xFD12345.LED.69.OFF\xFE" Unit="" Analog="true" Text="false" Sensor="false" SourceValHigh="100" DestValHigh="100"/>
	<CommCmd Title="6-fach Taster 12345 - Extern Led 6" Comment="" CmdOn="\xFD12345.LED.70.ON.&lt;v&gt;.0\xFE" CmdOff="\xFD12345.LED.70.OFF\xFE" Unit="" Analog="true" Text="false" Sensor="false" SourceValHigh="100" DestValHigh="100"/>
	<CommCmd Title="6-fach Taster 12345 - RFID Leser" Comment="" CmdOn="\xFD12345.RFD.65.TAG_ID.\v\xFE" CmdOff="" Unit="&lt;v.x&gt;" Analog="false" Text="true" Sensor="true" SourceValHigh="100" DestValHigh="100"/>
	<CommCmd Title="6-fach Taster 12345 - RFID Leser" Comment="" CmdOn="\xFD12345.RFD.66.TAG_ID.\v\xFE" CmdOff="" Unit="&lt;v.x&gt;" Analog="false" Text="true" Sensor="true" SourceValHigh="100" DestValHigh="100"/>
	<CommCmd Title="6-fach Taster 12345 - RFID Leser" Comment="" CmdOn="\xFD12345.RFD.67.TAG_ID.\v\xFE" CmdOff="" Unit="&lt;v.x&gt;" Analog="false" Text="true" Sensor="true" SourceValHigh="100" DestValHigh="100"/>
	<CommCmd Title="6-fach Taster 12345 - RFID Leser" Comment="" CmdOn="\xFD12345.RFD.68.TAG_ID.\v\xFE" CmdOff="" Unit="&lt;v.x&gt;" Analog="false" Text="true" Sensor="true" SourceValHigh="100" DestValHigh="100"/>
	<CommCmd Title="6-fach Taster 12345 - RFID Leser" Comment="" CmdOn="\xFD12345.RFD.69.TAG_ID.\v\xFE" CmdOff="" Unit="&lt;v.x&gt;" Analog="false" Text="true" Sensor="true" SourceValHigh="100" DestValHigh="100"/>
	</Comm>
*)
END_ACTION

END_FUNCTION_BLOCK

// ---- POUs/RS485_Hausbus_FB/Events/fb_BusTasterEvent.TcPOU
FUNCTION_BLOCK fb_BusTasterEvent
VAR_INPUT
	 I_sID         			:STRING(10);     // Geräte-ID (z.B. '12345')
	 I_sInstID				:STRING(2) 	:=	'17';
	 I_sReceivedString		:STRING(255);	
END_VAR
VAR_OUTPUT
	Q_bOut					:BOOL;
END_VAR
VAR
	findString0				:STRING ;
	findString1				:STRING ;
END_VAR


findString0 := CONCAT(I_sID,'.');
findString0 := CONCAT(findString0,'BTN');
findString0 := CONCAT(findString0,'.');
findString0 := CONCAT(findString0,I_sInstID);
findString0 := CONCAT(findString0,'.');
findString0 := CONCAT(findString0,'STATUS.0');

findString1 := CONCAT(I_sID,'.');
findString1 := CONCAT(findString1,'BTN');
findString1 := CONCAT(findString1,'.');
findString1 := CONCAT(findString1,I_sInstID);
findString1 := CONCAT(findString1,'.');
findString1 := CONCAT(findString1,'STATUS.1');

IF FIND(I_sReceivedString,findString0) >0 
THEN
	Q_bOut := FALSE;
ELSIF
	FIND(I_sReceivedString,findString1) >0 
THEN
	Q_bOut := TRUE;
END_IF

END_FUNCTION_BLOCK

// ---- POUs/RS485_Hausbus_FB/Events/fb_BusTempEvent.TcPOU
FUNCTION_BLOCK fb_BusTempEvent
VAR_INPUT
	 I_sID         			:STRING(10);     // Geräte-ID (z.B. '12345')
	 I_sInstID				:STRING(2) 	:=	'17';
	 I_sReceivedString		:STRING(255);	
	 I_bReset				:BOOL;
	 
END_VAR
VAR_OUTPUT
	Q_lrTemp				:LREAL;
END_VAR
VAR	
	findStringTemp			:STRING;	(* Wird für TMP/ BRS/ RHD verwendet *)

	sTemp1					:STRING;
	sTemp2					:STRING;
	
END_VAR

findStringTemp	:= CONCAT(I_sID,'.');
findStringTemp	:= CONCAT(findStringTemp,'TMP');
findStringTemp	:= CONCAT(findStringTemp,'.');
findStringTemp	:= CONCAT(findStringTemp,I_sInstID);
findStringTemp	:= CONCAT(findStringTemp,'.');

IF I_bReset
THEN
	sTemp1 := '0';
ELSE
	IF FIND(I_sReceivedString,findStringTemp) >0 
	THEN
		sTemp1 :=MID(I_sReceivedString, (* LÄNGE*) 4, FIND(I_sReceivedString,'TMP.1.STATUS.')+ LEN('TMP.1.STATUS.'));
	END_IF
END_IF

Q_lrTemp :=	STRING_TO_LREAL(sTemp1);

END_FUNCTION_BLOCK

// ---- POUs/RS485_Hausbus_FB/Events/fb_BusBrsEvent.TcPOU
FUNCTION_BLOCK fb_BusBrsEvent
VAR_INPUT
	 I_sID         			:STRING(10);     // Geräte-ID (z.B. '12345')
	 I_sInstID				:STRING(2) 	:=	'17';
	 I_sReceivedString		:STRING(255);	
	 I_bReset				:BOOL;
END_VAR
VAR_OUTPUT
	Q_lrBrs				:LREAL;
END_VAR
VAR	
	findStringTemp			:STRING;	(* Wird für TMP/ BRS/ RHD verwendet *)

	sBrs1					:STRING;
	sBrs2					:STRING;
	
END_VAR

findStringTemp	:= CONCAT(I_sID,'.');
findStringTemp	:= CONCAT(findStringTemp,'BRS');
findStringTemp	:= CONCAT(findStringTemp,'.');
findStringTemp	:= CONCAT(findStringTemp,I_sInstID);
findStringTemp	:= CONCAT(findStringTemp,'.');

IF I_bReset
THEN
	sBrs1 := '0';
ELSE
	IF FIND(I_sReceivedString,findStringTemp) >0 
	THEN
		sBrs1 :=MID(I_sReceivedString, (* LÄNGE*) 4, FIND(I_sReceivedString,'BRS.1.STATUS.')+ LEN('BRS.1.STATUS.'));
	END_IF
END_IF

Q_lrBrs :=	STRING_TO_LREAL(sBrs1);

END_FUNCTION_BLOCK

// ---- POUs/RS485_Hausbus_FB/Events/fb_BusRhdEvent.TcPOU
FUNCTION_BLOCK fb_BusRhdEvent
VAR_INPUT
	 I_sID         			:STRING(10);     // Geräte-ID (z.B. '12345')
	 I_sInstID				:STRING(2) 	:=	'17';
	 I_sReceivedString		:STRING(255);	
	 I_bReset				:BOOL;
END_VAR
VAR_OUTPUT
	Q_lrRhd					:LREAL;
END_VAR
VAR	
	findStringTemp			:STRING;	(* Wird für TMP/ BRS/ RHD verwendet *)

	sRhd1					:STRING;
	sRhd2					:STRING;
	
END_VAR

findStringTemp	:= CONCAT(I_sID,'.');
findStringTemp	:= CONCAT(findStringTemp,'RHD');
findStringTemp	:= CONCAT(findStringTemp,'.');
findStringTemp	:= CONCAT(findStringTemp,I_sInstID);
findStringTemp	:= CONCAT(findStringTemp,'.');

IF I_bReset
THEN
	sRhd1 := '0';
ELSE
	IF FIND(I_sReceivedString,findStringTemp) >0 
	THEN
		sRhd1 :=MID(I_sReceivedString, (* LÄNGE*) 4, FIND(I_sReceivedString,'RHD.1.STATUS.')+ LEN('RHD.1.STATUS.'));
	END_IF
END_IF

Q_lrRhd :=	STRING_TO_LREAL(sRhd1);

END_FUNCTION_BLOCK

// ---- POUs/RS485_Hausbus_FB/BusTaster/fb_StringConvTB6F.TcPOU
(*======================================================================================================================================*)
(*fb_StringConvTB6F:	Zusammensetzen des Strings für 6Fach Bust Taster (LEDs und Hintergrundbeleuchtung und Reset)*)
(*
Date          	| Version    	| created under        	| Author          	| Remark *)
(*====================================================================================================================================================*)
(*05/05/2025   	| 1.00      		| TC3		  		| N.Kersting       | first release *)
(*06/05/2025   	| 1.01      		| TC3		  		| N.Kersting       | Externe LEDs Nachgerüstet *)
(*08/05/2025   	| 1.02      		| TC3		  		| N.Kersting       | Umschaltung ob Externe LEDs verwendet werden oder nicht *)
(*====================================================================================================================================================*)
FUNCTION_BLOCK fb_StringConvTB6F
VAR_INPUT
	I_bReset			:BOOL;							(* Reset Befehl auslösen *)
	I_bExtLED			:BOOL;							(* Schaltet nur die Externen LEDs*)
	I_bSetBackground	:BOOL;							(* Nur Hintergrundbeleuchtung setzen *)
	I_bHasExtLED		:BOOL := FALSE;					(* Wenn Aktiv, werden Die Externen LEDs bei Hintergrundbeleuchtung mit gesendet! *)
	I_diID				:DINT;							(* Device ID *)
	I_iLED     	 		:ARRAY[1..6] OF INT;     	  	(* gewünschter LED-Zustand (TRUE = 100 %)*)
	I_iLEDExt  	 		:ARRAY[1..6] OF INT;     	  	(* gewünschter LED-Zustand (TRUE = 100 %)*)
	I_iLEDBg			:INT;							(* gewünschte Hintergrundbeleuchtung Achtung nur für Interne LEDs*)
	I_sStartZeichen		:BYTE := 16#FD;					(* Startzeichen Präfix *)
	I_sEndZeichen		:BYTE := 16#FE;					(* Endzeichen Suffix *)
END_VAR
VAR_OUTPUT
	Q_sConvString		:STRING(255);
END_VAR
VAR
	iStartInstID		:INT :=49;
	iStartLED			:INT := 1;
	
	iStartInstIDExt		:INT :=65;
	iStartLEDExt		:INT := 1;
END_VAR

IF NOT I_bReset
THEN
	IF I_bSetBackground
	THEN
		IF I_bHasExtLED
		THEN
			(* Externe LEDs*)
			iStartInstIDExt := 65;
			iStartLEDExt := 1;
			
			Q_sConvString:=	CONCAT(F_ToCHR(I_sStartZeichen),DINT_TO_STRING(I_diID));
			Q_sConvString:=	CONCAT(Q_sConvString,'.LED.');
			Q_sConvString:=	CONCAT(Q_sConvString,INT_TO_STRING(iStartInstIDExt));
			Q_sConvString:=	CONCAT(Q_sConvString,'.SET_MBR.');
			Q_sConvString:=	CONCAT(Q_sConvString,INT_TO_STRING(I_iLEDBg));
			Q_sConvString:=	CONCAT(Q_sConvString,F_ToCHR(I_sEndZeichen));
			
			iStartInstIDExt := iStartInstIDExt +1;
			iStartLEDExt := 	iStartLEDExt +1;
			
			Q_sConvString:=	CONCAT(Q_sConvString,F_ToCHR(I_sStartZeichen));
			Q_sConvString:=	CONCAT(Q_sConvString,DINT_TO_STRING(I_diID));
			Q_sConvString:=	CONCAT(Q_sConvString,'.LED.');
			Q_sConvString:=	CONCAT(Q_sConvString,INT_TO_STRING(iStartInstIDExt));
			Q_sConvString:=	CONCAT(Q_sConvString,'.SET_MBR.');
			Q_sConvString:=	CONCAT(Q_sConvString,INT_TO_STRING(I_iLEDBg));
			Q_sConvString:=	CONCAT(Q_sConvString,F_ToCHR(I_sEndZeichen));
			
			iStartInstIDExt := iStartInstIDExt +1;
			iStartLEDExt := 	iStartLEDExt +1;
			
			Q_sConvString:=	CONCAT(Q_sConvString,F_ToCHR(I_sStartZeichen));
			Q_sConvString:=	CONCAT(Q_sConvString,DINT_TO_STRING(I_diID));
			Q_sConvString:=	CONCAT(Q_sConvString,'.LED.');
			Q_sConvString:=	CONCAT(Q_sConvString,INT_TO_STRING(iStartInstIDExt));
			Q_sConvString:=	CONCAT(Q_sConvString,'.SET_MBR.');
			Q_sConvString:=	CONCAT(Q_sConvString,INT_TO_STRING(I_iLEDBg));
			Q_sConvString:=	CONCAT(Q_sConvString,F_ToCHR(I_sEndZeichen));
			
			iStartInstIDExt := iStartInstIDExt +1;
			iStartLEDExt := 	iStartLEDExt +1;
			
			Q_sConvString:=	CONCAT(Q_sConvString,F_ToCHR(I_sStartZeichen));
			Q_sConvString:=	CONCAT(Q_sConvString,DINT_TO_STRING(I_diID));
			Q_sConvString:=	CONCAT(Q_sConvString,'.LED.');
			Q_sConvString:=	CONCAT(Q_sConvString,INT_TO_STRING(iStartInstIDExt));
			Q_sConvString:=	CONCAT(Q_sConvString,'.SET_MBR.');
			Q_sConvString:=	CONCAT(Q_sConvString,INT_TO_STRING(I_iLEDBg));
			Q_sConvString:=	CONCAT(Q_sConvString,F_ToCHR(I_sEndZeichen));
			
			iStartInstIDExt := iStartInstIDExt +1;
			iStartLEDExt := 	iStartLEDExt +1;
			
			Q_sConvString:=	CONCAT(Q_sConvString,F_ToCHR(I_sStartZeichen));
			Q_sConvString:=	CONCAT(Q_sConvString,DINT_TO_STRING(I_diID));
			Q_sConvString:=	CONCAT(Q_sConvString,'.LED.');
			Q_sConvString:=	CONCAT(Q_sConvString,INT_TO_STRING(iStartInstIDExt));
			Q_sConvString:=	CONCAT(Q_sConvString,'.SET_MBR.');
			Q_sConvString:=	CONCAT(Q_sConvString,INT_TO_STRING(I_iLEDBg));
			Q_sConvString:=	CONCAT(Q_sConvString,F_ToCHR(I_sEndZeichen));
			
			iStartInstIDExt := iStartInstIDExt +1;
			iStartLEDExt := 	iStartLEDExt +1;
			
			Q_sConvString:=	CONCAT(Q_sConvString,F_ToCHR(I_sStartZeichen));
			Q_sConvString:=	CONCAT(Q_sConvString,DINT_TO_STRING(I_diID));
			Q_sConvString:=	CONCAT(Q_sConvString,'.LED.');
			Q_sConvString:=	CONCAT(Q_sConvString,INT_TO_STRING(iStartInstIDExt));
			Q_sConvString:=	CONCAT(Q_sConvString,'.SET_MBR.');
			Q_sConvString:=	CONCAT(Q_sConvString,INT_TO_STRING(I_iLEDBg));
			Q_sConvString:=	CONCAT(Q_sConvString,F_ToCHR(I_sEndZeichen));
			
			(* Interne LEDs*)
			(* Hintergrundbeleuchtung setzen *)
			
			Q_sConvString:=	CONCAT(Q_sConvString,F_ToCHR(I_sStartZeichen));
			Q_sConvString:=	CONCAT(Q_sConvString,DINT_TO_STRING(I_diID));
			Q_sConvString:=	CONCAT(Q_sConvString,'.LBN.');
			Q_sConvString:=	CONCAT(Q_sConvString,INT_TO_STRING(16));
			Q_sConvString:=	CONCAT(Q_sConvString,'.SET_MBR.');
			Q_sConvString:=	CONCAT(Q_sConvString,INT_TO_STRING(I_iLEDBg));
			Q_sConvString:=	CONCAT(Q_sConvString,F_ToCHR(I_sEndZeichen));
			
		ELSE
			(* Interne LEDs*)
			(* Hintergrundbeleuchtung setzen *)
			Q_sConvString:=	CONCAT(F_ToCHR(I_sStartZeichen),DINT_TO_STRING(I_diID));
			Q_sConvString:=	CONCAT(Q_sConvString,'.LBN.');
			Q_sConvString:=	CONCAT(Q_sConvString,INT_TO_STRING(16));
			Q_sConvString:=	CONCAT(Q_sConvString,'.SET_MBR.');
			Q_sConvString:=	CONCAT(Q_sConvString,INT_TO_STRING(I_iLEDBg));
			Q_sConvString:=	CONCAT(Q_sConvString,F_ToCHR(I_sEndZeichen));
		END_IF
	ELSE
		(* Normale Helligkeit setzen *)
		IF NOT I_bExtLED
		THEN
			(* Interne LEDs*)
			iStartInstID := 49;
			iStartLED := 1;
			
			Q_sConvString:=	CONCAT(F_ToCHR(I_sStartZeichen),DINT_TO_STRING(I_diID));
			Q_sConvString:=	CONCAT(Q_sConvString,'.LED.');
			Q_sConvString:=	CONCAT(Q_sConvString,INT_TO_STRING(iStartInstID));
			Q_sConvString:=	CONCAT(Q_sConvString,'.ON.');
			Q_sConvString:=	CONCAT(Q_sConvString,INT_TO_STRING(I_iLED[iStartLED]));
			Q_sConvString:=	CONCAT(Q_sConvString,F_ToCHR(I_sEndZeichen));
			
			iStartInstID := iStartInstID +1;
			iStartLED := 	iStartLED +1;
			
			Q_sConvString:=	CONCAT(Q_sConvString,F_ToCHR(I_sStartZeichen));
			Q_sConvString:=	CONCAT(Q_sConvString,DINT_TO_STRING(I_diID));
			Q_sConvString:=	CONCAT(Q_sConvString,'.LED.');
			Q_sConvString:=	CONCAT(Q_sConvString,INT_TO_STRING(iStartInstID));
			Q_sConvString:=	CONCAT(Q_sConvString,'.ON.');
			Q_sConvString:=	CONCAT(Q_sConvString,INT_TO_STRING(I_iLED[iStartLED]));
			Q_sConvString:=	CONCAT(Q_sConvString,F_ToCHR(I_sEndZeichen));
			
			iStartInstID := iStartInstID +1;
			iStartLED := 	iStartLED +1;
			
			Q_sConvString:=	CONCAT(Q_sConvString,F_ToCHR(I_sStartZeichen));
			Q_sConvString:=	CONCAT(Q_sConvString,DINT_TO_STRING(I_diID));
			Q_sConvString:=	CONCAT(Q_sConvString,'.LED.');
			Q_sConvString:=	CONCAT(Q_sConvString,INT_TO_STRING(iStartInstID));
			Q_sConvString:=	CONCAT(Q_sConvString,'.ON.');
			Q_sConvString:=	CONCAT(Q_sConvString,INT_TO_STRING(I_iLED[iStartLED]));
			Q_sConvString:=	CONCAT(Q_sConvString,F_ToCHR(I_sEndZeichen));
			
			iStartInstID := iStartInstID +1;
			iStartLED := 	iStartLED +1;
			
			Q_sConvString:=	CONCAT(Q_sConvString,F_ToCHR(I_sStartZeichen));
			Q_sConvString:=	CONCAT(Q_sConvString,DINT_TO_STRING(I_diID));
			Q_sConvString:=	CONCAT(Q_sConvString,'.LED.');
			Q_sConvString:=	CONCAT(Q_sConvString,INT_TO_STRING(iStartInstID));
			Q_sConvString:=	CONCAT(Q_sConvString,'.ON.');
			Q_sConvString:=	CONCAT(Q_sConvString,INT_TO_STRING(I_iLED[iStartLED]));
			Q_sConvString:=	CONCAT(Q_sConvString,F_ToCHR(I_sEndZeichen));
			
			iStartInstID := iStartInstID +1;
			iStartLED := 	iStartLED +1;
			
			Q_sConvString:=	CONCAT(Q_sConvString,F_ToCHR(I_sStartZeichen));
			Q_sConvString:=	CONCAT(Q_sConvString,DINT_TO_STRING(I_diID));
			Q_sConvString:=	CONCAT(Q_sConvString,'.LED.');
			Q_sConvString:=	CONCAT(Q_sConvString,INT_TO_STRING(iStartInstID));
			Q_sConvString:=	CONCAT(Q_sConvString,'.ON.');
			Q_sConvString:=	CONCAT(Q_sConvString,INT_TO_STRING(I_iLED[iStartLED]));
			Q_sConvString:=	CONCAT(Q_sConvString,F_ToCHR(I_sEndZeichen));
			
			iStartInstID := iStartInstID +1;
			iStartLED := 	iStartLED +1;
			
			Q_sConvString:=	CONCAT(Q_sConvString,F_ToCHR(I_sStartZeichen));
			Q_sConvString:=	CONCAT(Q_sConvString,DINT_TO_STRING(I_diID));
			Q_sConvString:=	CONCAT(Q_sConvString,'.LED.');
			Q_sConvString:=	CONCAT(Q_sConvString,INT_TO_STRING(iStartInstID));
			Q_sConvString:=	CONCAT(Q_sConvString,'.ON.');
			Q_sConvString:=	CONCAT(Q_sConvString,INT_TO_STRING(I_iLED[iStartLED]));
			Q_sConvString:=	CONCAT(Q_sConvString,F_ToCHR(I_sEndZeichen));
		ELSE
			(* Externe LEDs*)
			iStartInstIDExt := 65;
			iStartLEDExt := 1;
			
			Q_sConvString:=	CONCAT(F_ToCHR(I_sStartZeichen),DINT_TO_STRING(I_diID));
			Q_sConvString:=	CONCAT(Q_sConvString,'.LED.');
			Q_sConvString:=	CONCAT(Q_sConvString,INT_TO_STRING(iStartInstIDExt));
			Q_sConvString:=	CONCAT(Q_sConvString,'.ON.');
			Q_sConvString:=	CONCAT(Q_sConvString,INT_TO_STRING(I_iLEDExt[iStartLEDExt]));
			Q_sConvString:=	CONCAT(Q_sConvString,F_ToCHR(I_sEndZeichen));
			
			iStartInstIDExt := iStartInstIDExt +1;
			iStartLEDExt := 	iStartLEDExt +1;
			
			Q_sConvString:=	CONCAT(Q_sConvString,F_ToCHR(I_sStartZeichen));
			Q_sConvString:=	CONCAT(Q_sConvString,DINT_TO_STRING(I_diID));
			Q_sConvString:=	CONCAT(Q_sConvString,'.LED.');
			Q_sConvString:=	CONCAT(Q_sConvString,INT_TO_STRING(iStartInstIDExt));
			Q_sConvString:=	CONCAT(Q_sConvString,'.ON.');
			Q_sConvString:=	CONCAT(Q_sConvString,INT_TO_STRING(I_iLEDExt[iStartLEDExt]));
			Q_sConvString:=	CONCAT(Q_sConvString,F_ToCHR(I_sEndZeichen));
			
			iStartInstIDExt := iStartInstIDExt +1;
			iStartLEDExt := 	iStartLEDExt +1;
			
			Q_sConvString:=	CONCAT(Q_sConvString,F_ToCHR(I_sStartZeichen));
			Q_sConvString:=	CONCAT(Q_sConvString,DINT_TO_STRING(I_diID));
			Q_sConvString:=	CONCAT(Q_sConvString,'.LED.');
			Q_sConvString:=	CONCAT(Q_sConvString,INT_TO_STRING(iStartInstIDExt));
			Q_sConvString:=	CONCAT(Q_sConvString,'.ON.');
			Q_sConvString:=	CONCAT(Q_sConvString,INT_TO_STRING(I_iLEDExt[iStartLEDExt]));
			Q_sConvString:=	CONCAT(Q_sConvString,F_ToCHR(I_sEndZeichen));
			
			iStartInstIDExt := iStartInstIDExt +1;
			iStartLEDExt := 	iStartLEDExt +1;
			
			Q_sConvString:=	CONCAT(Q_sConvString,F_ToCHR(I_sStartZeichen));
			Q_sConvString:=	CONCAT(Q_sConvString,DINT_TO_STRING(I_diID));
			Q_sConvString:=	CONCAT(Q_sConvString,'.LED.');
			Q_sConvString:=	CONCAT(Q_sConvString,INT_TO_STRING(iStartInstIDExt));
			Q_sConvString:=	CONCAT(Q_sConvString,'.ON.');
			Q_sConvString:=	CONCAT(Q_sConvString,INT_TO_STRING(I_iLEDExt[iStartLEDExt]));
			Q_sConvString:=	CONCAT(Q_sConvString,F_ToCHR(I_sEndZeichen));
			
			iStartInstIDExt := iStartInstIDExt +1;
			iStartLEDExt := 	iStartLEDExt +1;
			
			Q_sConvString:=	CONCAT(Q_sConvString,F_ToCHR(I_sStartZeichen));
			Q_sConvString:=	CONCAT(Q_sConvString,DINT_TO_STRING(I_diID));
			Q_sConvString:=	CONCAT(Q_sConvString,'.LED.');
			Q_sConvString:=	CONCAT(Q_sConvString,INT_TO_STRING(iStartInstIDExt));
			Q_sConvString:=	CONCAT(Q_sConvString,'.ON.');
			Q_sConvString:=	CONCAT(Q_sConvString,INT_TO_STRING(I_iLEDExt[iStartLEDExt]));
			Q_sConvString:=	CONCAT(Q_sConvString,F_ToCHR(I_sEndZeichen));
			
			iStartInstIDExt := iStartInstIDExt +1;
			iStartLEDExt := 	iStartLEDExt +1;
			
			Q_sConvString:=	CONCAT(Q_sConvString,F_ToCHR(I_sStartZeichen));
			Q_sConvString:=	CONCAT(Q_sConvString,DINT_TO_STRING(I_diID));
			Q_sConvString:=	CONCAT(Q_sConvString,'.LED.');
			Q_sConvString:=	CONCAT(Q_sConvString,INT_TO_STRING(iStartInstIDExt));
			Q_sConvString:=	CONCAT(Q_sConvString,'.ON.');
			Q_sConvString:=	CONCAT(Q_sConvString,INT_TO_STRING(I_iLEDExt[iStartLEDExt]));
			Q_sConvString:=	CONCAT(Q_sConvString,F_ToCHR(I_sEndZeichen));
		END_IF
	END_IF
ELSE
	(* Reset *)
	Q_sConvString:=	CONCAT(F_ToCHR(I_sStartZeichen),DINT_TO_STRING(I_diID));
	Q_sConvString:=	CONCAT(Q_sConvString,'.SYS.');
	Q_sConvString:=	CONCAT(Q_sConvString,INT_TO_STRING(1));
	Q_sConvString:=	CONCAT(Q_sConvString,'.RESET');
	Q_sConvString:=	CONCAT(Q_sConvString,F_ToCHR(I_sEndZeichen));
END_IF

END_FUNCTION_BLOCK

// ---- POUs/RS485_Hausbus_FB/RS485 COM/fb_RS485ComCheck.TcPOU
(*======================================================================================================================================*)
(*fb_RS485ComCheck:	Einfacher Universal Ping Baustein um von allerlei Geräten von haus-bus.de Kommunikation zu Checken über RS485 
	In Diesem Fall ist es für einen Taster (BTN) bei einem Relais sollte es (OUT) sein*)
(*
Date          	| Version    	| created under        	| Author          	| Remark *)
(*====================================================================================================================================================*)
(*05/05/2025   	| 1.00      		| TC3		  		| N.Kersting       | first release *)
(*06/05/2025   	| 1.01      		| TC3		  		| N.Kersting       | Bugfix Timeouts werden besser ausgewertet *)
(*07/05/2025   	| 1.02      		| TC3		  		| N.Kersting       | Bug in Schritt 2 behoben (weiter, wenn nicht Busy) *)
(*09/05/2025   	| 1.03      		| TC3		  		| N.Kersting       | Counter für verbindungsversuche inkl. erneut senden *)
(*10/05/2025   	| 1.04      		| TC3		  		| N.Kersting       | Umrüstung Auf Externen Fifo  *)
(*12/05/2025   	| 1.05      		| TC3		  		| N.Kersting       | Verriegelung über I_bStart, damit nich gesendet werden kann wenn nicht Freigegeben  *)
(*14/05/2025   	| 1.06      		| TC3		  		| N.Kersting       | Ausgänge ergänzt für Done  *)
(*====================================================================================================================================================*)
FUNCTION_BLOCK fb_RS485ComCheck
VAR_INPUT
	I_FifoID			:INT;
	I_bExecute			:BOOL;							(* Aktiviert den Baustein *)
	I_bStart			:BOOL;							(* Startet das Senden des Pings *)
	I_tPingIntervall	:TIME := T#5S;					(* Intervall Zeit wann die Kommunikation geprüft werden soll *)
	I_tPingTimeout		:TIME := T#2S;					(* Zeit, bis der Ping zurück gekommen sein muss *)
	I_diID				:DINT;							(* Device ID *)
	I_sPingSymbol		:STRING :='.BTN.';				(* Symbol, welches als Ping genutzt werden soll *)
	I_iInstID			:INT := 17;						(* Instanz ID *)
	I_sStartZeichen		:BYTE := 16#FD;					(* Startzeichen Präfix *)
	I_sEndZeichen		:BYTE := 16#FE;					(* Endzeichen Suffix *)
	I_StringReceived	:STRING(255);					(* Empfangener String *)
	I_iMaxPingTry		:INT := 5;
	I_bTasterMode		:BOOL;							(* Wenn ein Taster Abgefragt wird, gibt es die Besonderheit, dass dieser Selbst Signale Sendet (Helligkeit, temperatur usw. *)
END_VAR
VAR_OUTPUT
	Q_sSend				:STRING(255);
	Q_bBusy 			:BOOL;
	Q_bSendDone			:BOOL;
	Q_sState			:STRING;
	Q_bComOk			:BOOL;
	Q_bTimeout			:BOOL;
	Q_bError			:BOOL;
END_VAR
VAR
	sStringSend			:STRING;
	fbBusPingEvent		:ARRAY[1..6] OF fb_BusPingEvent;
	
	tonIntervall		:ton;
	tonTimeout			:ton;
	tonRecevieAutoReset	:ton;
	
	iStepReceive		:INT;
	iStep				:INT;
	icntComTry			:INT;
	iMaxComTry			:INT := 5;
	i					:INT;
	icntSymbole			:INT;
	
	bSend				:BOOL;
	bReceived			:BOOL;
	bCOMMem				:BOOL;
END_VAR

iMaxComTry :=	I_iMaxPingTry;

(* Intervall timer *)
tonIntervall(
	PT := I_tPingIntervall);
	
(* Timeout timer *)
tonTimeout(
	PT := I_tPingTimeout);
	
(* Ping String ertsllen *)
sStringSend:=	CONCAT(F_ToCHR(I_sStartZeichen),DINT_TO_STRING(I_diID));
sStringSend:=	CONCAT(sStringSend,I_sPingSymbol);
sStringSend:=	CONCAT(sStringSend,INT_TO_STRING(I_iInstID));
sStringSend:=	CONCAT(sStringSend,'.gSTATUS');
sStringSend:=	CONCAT(sStringSend,F_ToCHR(I_sEndZeichen));

IF NOT I_bExecute 
	AND NOT I_bTasterMode
THEN
	Q_bComOk := FALSE;
	Q_bTimeout := FALSE;
	tonIntervall.IN := FALSE;
	tonTimeout.IN := FALSE;
	sStringSend:= '';
	bSend := FALSE;
	iStep := 0;
ELSE
	ac01_Send();
END_IF

ACTION ac01_Send:
(* Sende Schrittkette *)
			
CASE iStep OF
(*=========================================================*)	
0:	Q_sState := ' INIT';
	tonIntervall.IN := FALSE;
	tonTimeout.IN := FALSE;
	bCOMMem := FALSE;
	bSend := FALSE;
	Q_bBusy := FALSE;
	Q_sSend := '';
	
	IF I_bExecute
		AND I_bStart
	THEN
		Q_bSendDone := FALSE;
		Q_bBusy := TRUE;
		iStep := iStep +1;
	ELSIF
		NOT I_bExecute
		AND I_bTasterMode
	THEN
		iStep := 10;
	END_IF

(*=========================================================*)	
1:	Q_sState := 'Starte Sendebefehl';
	
	IF GVL_RS485FiFoSend.bSendDoneFiFo[I_FifoID]
	THEN
		tonTimeout.IN := TRUE;
		Q_sSend := sStringSend;
	END_IF
	IF NOT GVL_RS485FiFoSend.bSendDoneFiFo[I_FifoID]
	THEN
		tonTimeout.IN := FALSE;
		iStep := iStep +1;
	ELSIF
		tonTimeout.Q
	THEN
		tonTimeout.IN := FALSE;
		Q_sState := 'Timeout Send Busy';
		iStep := -1;
	END_IF
	
(*=========================================================*)	
2:	Q_sState := 'Auswertung Senden';
	bSend := FALSE;	
	tonTimeout.IN := TRUE;
	
	IF GVL_RS485FiFoSend.bSendDoneFiFo[I_FifoID]
	THEN
		Q_sSend := '';
		Q_bSendDone := TRUE;
		tonTimeout.IN := FALSE;
		iStep := iStep +1;
	ELSIF
		tonTimeout.Q
	THEN
		Q_sState := 'Timeout Send Done';
		iStep := -2;
	END_IF
		
(*=========================================================*)	
3:	Q_sState := 'Warte auf Empfang';
	tonTimeout.IN := TRUE;
	
	IF tonTimeout.Q
	THEN
		(* Kommunikations versuche *)
		IF icntComTry <iMaxComTry
		THEN
			icntComTry := icntComTry +1;
			iStep := 5;				(* Erneut Senden *)
		ELSE
			Q_sState := 'Timeout kein Ping Empfangen';
			Q_bComOk := FALSE;
			Q_bTimeout := TRUE;
			iStep := -4;	(* Erneut Empfangen *)
		END_IF
	ELSE
		
		IF	bCOMMem
		THEN
			bCOMMem := FALSE;
			iStep := iStep+1;		(* Telegram erhalten *)
		END_IF
	END_IF
	
(*=========================================================*)	
4:	Q_sState := 'Ping Empfangen, Warte auf Intervall';
	tonIntervall.IN := TRUE;
	Q_bComOk := TRUE;
	Q_bTimeout := FALSE;
	
	IF tonIntervall.Q
		AND I_bStart
	THEN
		icntComTry := 0;	(* Wenn die Verbindung wieder da ist dürfen die Versuche gelöscht werden *)
		iStep := 0;
	END_IF

(*=========================================================*)	
5:	Q_sState := 'Ping nicht Empfangen, Warte auf Intervall';
	tonIntervall.IN := TRUE;
	
	IF tonIntervall.Q
		AND I_bStart
	THEN
		iStep := 0;
	END_IF

(*=========================================================*)	
10:	Q_sState := 'Warten Auf Automatischen Ping vom Taster';
	tonIntervall.IN := TRUE;
	
	IF tonIntervall.Q
		AND I_bStart
	THEN
		Q_bComOk := FALSE;
		iStep := 0;
	ELSE
		IF bCOMMem
		THEN
			tonIntervall.IN := FALSE;
			Q_bComOk := TRUE;
			iStep := 0;
		END_IF
	END_IF	
ELSE
	tonIntervall.IN := TRUE;
	tonTimeout.IN := FALSE;
	Q_bComOk := FALSE;
	bSend := FALSE;
	Q_bBusy := FALSE;
	icntComTry := 0;
	Q_sSend := '';
	
	IF tonIntervall.Q
		AND I_bStart
	THEN
		iStep := 0;
	END_IF
END_CASE

IF I_bTasterMode
THEN
	icntSymbole := 0;
	(* Durchgehend Checken ob Ping kommt *)
	FOR i := 1 TO 6 BY 1 DO 
		fbBusPingEvent[i](
			I_bReset := 			FALSE,
			I_sID:= 				DINT_TO_STRING(I_diID ), 
			I_iInstID:=				I_iInstID -1 +i,	
			I_sReceivedString:= 	I_StringReceived, 
			I_bTasterMode := 		TRUE,
			Q_bOut=> 				);
			
		IF fbBusPingEvent[i].Q_bOut
		THEN
			icntSymbole := icntSymbole +1;
		END_IF
	END_FOR
	
	IF iStep > 0
		AND icntSymbole >0
	THEN
		bCOMMem := TRUE;
	END_IF
ELSE
	(* Nur nach der einen ID Gucken *)
	fbBusPingEvent[1](
		I_bReset := 			FALSE,
		I_sID:= 				DINT_TO_STRING(I_diID ), 
		I_iInstID:=				I_iInstID,	
		I_sReceivedString:= 	I_StringReceived, 
		I_bTasterMode := 		FALSE,
		Q_bOut=> 				);
		
	IF iStep > 0
		AND fbBusPingEvent[1].Q_bOut
	THEN
		bCOMMem := TRUE;
	END_IF
END_IF
END_ACTION

END_FUNCTION_BLOCK

// ---- POUs/RS485_Hausbus_FB/Events/fb_BusPingEvent.TcPOU
FUNCTION_BLOCK fb_BusPingEvent
VAR_INPUT
	 I_sID         			:STRING(10);     // Geräte-ID (z.B. '12345')
	 I_sReceivedString		:STRING(255);	
	 I_iInstID				:INT := 17;						(* Instanz ID *)
	 I_bTasterMode			:BOOL;
	 I_bReset				:BOOL;
END_VAR
VAR_OUTPUT
	Q_bOut					:BOOL;
END_VAR
VAR
	findString0				:STRING ;
	findString1				:STRING ;
	findString2				:STRING ;
	findString3				:STRING ;
	findString4				:STRING ;
	
END_VAR


findString0 := CONCAT(I_sID,'.');
findString0 := CONCAT(findString0,'BTN');
findString0 := CONCAT(findString0,'.');
findString0 := CONCAT(findString0,INT_TO_STRING(I_iInstID));
findString0 := CONCAT(findString0,'.');
findString0 := CONCAT(findString0,'rSTATUS');

(* Wenn ein Taster gedrückt wird *)
findString1 := CONCAT(I_sID,'.');
findString1 := CONCAT(findString1,'BTN');
findString1 := CONCAT(findString1,'.');
findString1 := CONCAT(findString1,INT_TO_STRING(I_iInstID));
findString1 := CONCAT(findString1,'.');
findString1 := CONCAT(findString1,'STATUS');

(* Wenn Ein Temperatur Event Kommt *)
findString2 := CONCAT(I_sID,'.');
findString2 := CONCAT(findString2,'TEMP.1.STATUS');
(* Wenn Ein Feuchtigkeit Event Kommt *)
findString3 := CONCAT(I_sID,'.');
findString3 := CONCAT(findString3,'RHD.1.STATUS');
(* Wenn Ein Helligkeit Event Kommt *)
findString4 := CONCAT(I_sID,'.');
findString4 := CONCAT(findString4,'BRS.1.STATUS');

IF I_bReset
THEN
	Q_bOut := FALSE;
ELSE
	IF FIND(I_sReceivedString,findString0) >0 
		OR (FIND(I_sReceivedString,findString1) >0 
		AND I_bTasterMode)
		OR (FIND(I_sReceivedString,findString2) >0 
		AND I_bTasterMode)
		OR (FIND(I_sReceivedString,findString3) >0 
		AND I_bTasterMode)
		OR (FIND(I_sReceivedString,findString4) >0 
		AND I_bTasterMode)
		
	THEN
		Q_bOut := TRUE;
	ELSE
		Q_bOut := FALSE;
	END_IF
END_IF

END_FUNCTION_BLOCK

// ---- POUs/RS485_Hausbus_FB/RelaisModul/fb_RelaisBus16F.TcPOU
(*======================================================================================================================================*)
(*fb_RelaisBus16F:		Einfache RS485 Kommunikation für Haus-bus.de Komponenten zum testen 	
						 *)
(*
Date          	| Version    	| created under        	| Author          	| Remark *)
(*====================================================================================================================================================*)
(*08/05/2025   	| 1.00      		| TC3		  		| N.Kersting       	| first release *)
(*08/05/2025   	| 1.01      		| TC3		  		| N.Kersting       	| Relais in Sections aufgeteilt um String Länge zu verringern *)
(*09/05/2025   	| 1.02      		| TC3		  		| N.Kersting       	| Ping Versuche Implementiert mit Globalen Parametern *)
(*10/05/2025   	| 2.00      		| TC3		  		| N.Kersting      	| Umstellung auf Externe FiFo Sendebaustein *)
(*12/05/2025   	| 2.01      		| TC3		  		| N.Kersting      	| Verriegelung für ComCheck hinzugefügt und Relais Sections auf 2 redzuziert *)
(*13/05/2025   	| 3.00      		| TC3		  		| N.Kersting       	| Viele Bugs gefixt, bei Änderung der Ausgängen wird nun eine Anforderung gesetzt  *)
(*====================================================================================================================================================*)
FUNCTION_BLOCK fb_RelaisBus16F
VAR_INPUT
	I_FifoID			:INT;
	I_bPingStart		:BOOL;						(* Ping Done vom Vorheriegen*)
	I_stInput			:ST_BusRelais16F_Input;
	I_StringReceived	:STRING(255);
END_VAR
VAR_OUTPUT
	Q_sFiFoSend			:STRING(255);
   	Q_stOutput			:ST_BusRelais16F_Output;
	Q_stCnt				:ST_BusRelais16F_Cnt;
END_VAR
VAR
(*----------------------------------------------*)
(* Interne Parameter*)
(*----------------------------------------------*)		
	bSetExecute			:BOOL := TRUE;				(* Aktiviert die Schrittketten, welche Telegramme versenden *)
	bCheckPing			:BOOL := TRUE;				(* Ping Checken Schrittkette Aktivieren *)
	sStartZeichen		:BYTE := 16#FD;				(* Startzeichen Präfix *)
	sEndZeichen			:BYTE := 16#FE;				(* Endzeichen Suffix *)
	iAnzResetSend		:INT := 2;					(* Anzahl der Sendeversuche bei Reset *)
	tPingTimer			:TIME:= T#5S;				(* Zeit, bis wiederholend der Ping versendet wird *)
	tReceiveTimeout		:TIME:= T#2S;				(* Zeit, bis die Event Schrittkette für das Empfangen Automatisch neu Startet*)
	tStartupLEDOn		:TIME:= T#3S;				(* Zeit, wie Lange die LEDS beim Startup kurz eingeschaltet werden *)
	tResetTimeout		:TIME:= T#8S;				(* Zeit, bis bei einem Reset es zu einem Fehler kommt, wenn kein Ping empfangen wird *)
	tResetReboot		:TIME:= T#3S;				(* Zeit, die nach einem Reset Abgewaretet wird damit das Gerät neustarten kann*)
	tResetStartup		:TIME:= T#1S;				(* Zeit, die nach einem Reset Abgewaretet wird bis ein Startup ausgeführt wird nach dem erhalt des Pings vom Gerät*)
	tStartupAfterReset	:TIME := T#5S;				(* Zeit, wann das Startup Zurückgesetzt wird, wenn der Ping verloren wird *)
(*----------------------------------------------*)
(* Strings *)
(*----------------------------------------------*)			
	sSendString			:STRING(255);
	sFiFoSend			:STRING(255);
	sReceived			:STRING(255);
	sLastSendString		:STRING(255);
	sLastSendString1	:STRING(255);
	sStateReset			:STRING;
(*----------------------------------------------*)
(* Funktionsbausteine *)
(*----------------------------------------------*)
	fbBusTasterEvent	:ARRAY[1..8] OF fb_BusTasterEvent;		(* Interne 8 Taster Abfragen *)
	fbStringConvR1B6F	:fb_StringConvRB16F;
	fbRS485ComCheck		:fb_RS485ComCheck;
(*----------------------------------------------*)
(* Indexe *)
(*----------------------------------------------*)	
	iDeviceStartup		:INT :=0;	(* Startup Schrittkette *)
	sDeviceStartup		:STRING;
    iState     			:INT := 0;
	iStepSet			:INT;
	i,h,j,l				:INT;
	idxLED				:INT;
	idxBtn				:INT := 1;
	ibOutMem			:ARRAY[1..16] OF BOOL;
	ibOutAnf			:ARRAY[1..16] OF BOOL;
	cntChangesOut		:INT;
	icntResetSend		:INT;
	iSection			:INT :=1;
	iMaxPingTry			:INT := 5;
(*----------------------------------------------*)
(* Timer/Trigger *)
(*----------------------------------------------*)		
	r_trigStartupAfterReset	:r_trig;
	r_TrigReset				:r_trig;		
	r_TrigCountBtn			:ARRAY[1..16] OF r_trig;
	
	tonStartupAfterReset	:ton;
	tonReceiveTimeout		:ton;
	tonResetTimeout			:ton;
	tonResetDone			:ton;
	tonStepStartup			:ton;
(*----------------------------------------------*)
(* Status *)
(*----------------------------------------------*)			
	bPingOK					:BOOL;
	bErrorEvent				:BOOL;
	bErrorPing				:BOOL;
	bErrorSet				:BOOL;
	bErrorReset				:BOOL;
	bResetBusy				:BOOL;
	bResetDone				:BOOL;
	bResetAutoStart			:BOOL;
	bStartupStart			:BOOL;
	bStartupDone			:BOOL;	
	bMemExt					:BOOL;
	bStartUpCheckPing		:BOOL;
	bActivateSend			:BOOL;
	bReadyToPing			:BOOL;
	bPingFreigabe			:BOOL;
	bSendeAnforderung		:BOOL;
END_VAR

(*============================================================================================*)
(* Parameter *)
tPingTimer :=		GVL_HausBus_Parameter.cTimePingTimeRelais;
tReceiveTimeout :=	GVL_HausBus_Parameter.cTimeReceiveTimeoutRelais;
bCheckPing :=		GVL_HausBus_Parameter.bUseRelaisPing;
iMaxPingTry :=		GVL_HausBus_Parameter.cMaxPingTry;

(*============================================================================================*)
(* Startup Zurücksetzen Reset *)
r_TrigReset(CLK := I_stInput.bReset);

(* Startup Zurücksetzen bei Busverlust *)
tonStartupAfterReset(
	IN := NOT bPingOK
			AND bCheckPing,
	PT:= tStartupAfterReset);

r_trigStartupAfterReset
	(CLK := tonStartupAfterReset.Q);
	
IF NOT I_stInput.bExecute
	OR r_TrigReset.Q
	OR r_trigStartupAfterReset.Q
THEN
	iDeviceStartup := 0;
END_IF

(*============================================================================================*)
(* Ping Dauerhaft Senden*)
ac02_Ping();
	
(*============================================================================================*)
(* Startup Schrittkette *)
CASE iDeviceStartup OF
(*============================================================================================*)
0: 	sDeviceStartup := 'INIT';
	bResetDone := FALSE;
	bStartupDone := FALSE;
	bStartupStart := FALSE;
	bResetAutoStart := FALSE;
	bStartUpCheckPing := FALSE;
	bActivateSend := FALSE;
	bReadyToPing := TRUE;
	bPingFreigabe := FALSE;
	
	iStepSet := 0;
	
	IF 	I_stInput.bExecute
	THEN
		iDeviceStartup := iDeviceStartup+1;
	END_IF
(*============================================================================================*)
1: 	sDeviceStartup := 'Device ID Prüfen';
	
	IF  I_stInput.diID <> 0
	THEN
		iDeviceStartup := iDeviceStartup+1;
	ELSE
		sDeviceStartup := 'ERROR- Device ID Prüfen';
	END_IF
(*============================================================================================*)
2: 	sDeviceStartup := 'Verbindung Prüfen';
	bStartUpCheckPing := TRUE;
	bPingFreigabe := TRUE;
	bActivateSend := TRUE;	(* Senden Aktivieren *)
	
	sDeviceStartup := CONCAT(sDeviceStartup,fbRS485ComCheck.Q_sState);
	
	IF fbRS485ComCheck.Q_bComOk
		OR NOT bCheckPing
	THEN
		iDeviceStartup := iDeviceStartup+1;
	END_IF

(*============================================================================================*)
3: 	sDeviceStartup := 'Reset Ausführen';	
	bActivateSend := TRUE;	(* Senden Aktivieren *)
	
	(*	RESET Device *)
	ac01_SetReset();
	bResetAutoStart := TRUE;
	
	sDeviceStartup :=	CONCAT(sDeviceStartup,sStateReset);
	
	IF bResetDone
	THEN
		iStepSet := 0;
		iDeviceStartup := iDeviceStartup+1;
	END_IF

(*============================================================================================*)
4: 	sDeviceStartup := 'Startup Ausführen';
		
	(* LED Setzen *)
	ac01_SetOutput();
	
	bStartupStart := TRUE;
	
	IF bStartupDone 
	THEN
		bStartupStart := FALSE;
		iDeviceStartup := 999;
	END_IF

(*============================================================================================*)
999: 
	(*bReadyToPing := NOT fbRS485SendCmd.Q_bBusy;*)
	
	(* LED Setzen *)
	ac01_SetOutput();
	
	(* Events Auslesen *)
	ac00_Event();
	
	(* Zähler *)
	ac10_Counter();
	
	sDeviceStartup := 'Startup Ausgeführt- Gerät im OP';
	
END_CASE

(*============================================================================================*)
(* Sendebaustein *)
IF bActivateSend
THEN
	IF fbRS485ComCheck.Q_sSend <>''
	THEN
		Q_sFiFoSend :=	fbRS485ComCheck.Q_sSend;
	ELSE
		Q_sFiFoSend :=	sFiFoSend;
	END_IF
END_IF

(*============================================================================================*)	
(* Zähler *)
ac10_Counter();
	
(*============================================================================================*)
(* Outputs *)
Q_stOutput.bCOM :=		bPingOK;

Q_stOutput.bError := 	bErrorEvent
						OR bErrorPing
						OR bErrorSet
						OR (NOT bPingOK
						AND bCheckPing);
						
Q_stOutput.bStartupDone	:=	bStartupDone;

Q_stOutput.sState :=	CONCAT(I_stInput.sName,'| ');
Q_stOutput.sState :=	CONCAT(Q_stOutput.sState, sDeviceStartup);

ACTION ac00_Event:
(*============================================================================================*)
(*	EVENT Schrittkette *)
(*============================================================================================*)
sReceived := I_StringReceived;
	
FOR i := 1 TO 8 BY 1 DO 
	fbBusTasterEvent[i](
		I_sID:= 				DINT_TO_STRING(I_stInput.diID), 
		I_sInstID:= 			INT_TO_STRING(i+96), 
		I_sReceivedString:= 	sReceived, 
		Q_bOut=> 				Q_stOutput.bInputs[i]);
END_FOR
END_ACTION

ACTION ac01_SetOutput:
(*============================================================================================*)
(*	LED Helligkeit Setzen/ Startup Schrittkette *)
(*============================================================================================*)

(* Einfaches Setzen der LED Helligkeiten (0-100 Prozent *)
(* Neu, es werden alle LEDs zu einem String zusammengefügt und Gleichzeitig gesetzt *)
tonStepStartup(
	PT:= tStartupLEDOn);

cntChangesOut := 0;
FOR l := 1 TO 16 BY 1 DO
	IF ibOutMem[l] <> I_stInput.bOut[l]
	THEN
		cntChangesOut := cntChangesOut +1;
	END_IF
END_FOR
	
CASE iStepSet OF
(*============================================================================================*)
0:	(* INIT und warten auf Change *)
	tonStepStartup.IN := FALSE;
	bPingFreigabe := TRUE; 
	iSection := 1;
	
	(* Merken ob eine Anforderung Ansteht *)
	IF cntChangesOut <>0
	THEN
		bSendeAnforderung := TRUE;
		FOR h := 1 TO 16 BY 1 DO
			ibOutAnf[h] := I_stInput.bOut[h];
		END_FOR
	END_IF
	
	IF (bSendeAnforderung
		AND bSetExecute)
		AND NOT bStartupStart
		AND fbRS485ComCheck.Q_sSend =''
	THEN
		bSendeAnforderung := FALSE;
		bPingFreigabe := FALSE; 
		(* Angeforderten Relaiszustand speichern *)
		FOR h := 1 TO 16 BY 1 DO
			ibOutMem[h] := I_stInput.bOut[h];
		END_FOR
		iStepSet := 10;
	ELSIF
		bStartupStart
	THEN
		iStepSet := 100;	(* Startup *)
	END_IF
	
(*============================================================================================*)
10:	(* String senden *)	
	(* Nur Relais Schreiben *)
	
	fbStringConvR1B6F(
		I_bReset:= 			FALSE, 
		I_bRedLEDOn:= 		FALSE, 
		I_bRedLEDOff:= 		FALSE, 
		I_iSection :=		iSection,
		I_diID:= 			I_stInput.diID, 
		I_bOut:= 			ibOutAnf, 
		I_sStartZeichen:= 	sStartZeichen, 
		I_sEndZeichen:= 	sEndZeichen,	 
		Q_sConvString=> 	sSendString);
		
	(* Senden an FiFo*)
	IF GVL_RS485FiFoSend.bSendDoneFiFo[I_FifoID]
	THEN
		sFiFoSend :=	sSendString;
	END_IF
	IF NOT GVL_RS485FiFoSend.bSendDoneFiFo[I_FifoID]
	THEN
		IF iSection <= 2
		THEN
			iSection :=	iSection+1;
		END_IF
		
		iStepSet := 20;
	END_IF
		
(*============================================================================================*)	
20:	(* Warten bis nicht Busy *)	
	IF GVL_RS485FiFoSend.bSendDoneFiFo[I_FifoID]	
	THEN
		sFiFoSend := ''; 
		
		IF iSection <= 2
		THEN
			sLastSendString :=	sSendString;
			iStepSet := 10;
		ELSE
			sLastSendString1 :=	sSendString;
			iStepSet := 0;
		END_IF
	END_IF
	
(*============================================================================================*)	
(* Startup  *)
100:	tonStepStartup.IN := TRUE;
	
	IF tonStepStartup.Q
	THEN
		iStepSet := 110;
	END_IF
	
(*============================================================================================*)
110:(* String senden *)	(* Alle Relais Ausschalten *)
	tonStepStartup.IN := FALSE;
		
	fbStringConvR1B6F(
		I_bReset:= 			FALSE, 
		I_bRedLEDOn:= 		FALSE, 
		I_bRedLEDOff:= 		FALSE, 
		I_iSection :=		iSection,
		I_diID:= 			I_stInput.diID, 
		I_bOut:= 			I_stInput.bOut, 
		I_sStartZeichen:= 	sStartZeichen, 
		I_sEndZeichen:= 	sEndZeichen,	 
		Q_sConvString=> 	sSendString);
		
	IF GVL_RS485FiFoSend.bSendDoneFiFo[I_FifoID]
	THEN
		sFiFoSend :=	sSendString;
	END_IF
	IF NOT GVL_RS485FiFoSend.bSendDoneFiFo[I_FifoID]
	THEN
		IF iSection <= 2
		THEN
			iSection :=	iSection+1;
		END_IF
		
		iStepSet := 111;
	END_IF
	
(*============================================================================================*)
111:(* String senden *)
	IF GVL_RS485FiFoSend.bSendDoneFiFo[I_FifoID]
	THEN
		sLastSendString :=	sSendString;
		sFiFoSend := ''; 
		
		IF iSection <= 2
		THEN
			iStepSet := 110;
		ELSE
			iStepSet := 112;
		END_IF
	END_IF
	
(*============================================================================================*)
112:(* String senden *)	(* Rote LED Einschalten *)
	tonStepStartup.IN := FALSE;
		
	fbStringConvR1B6F(
		I_bReset:= 			FALSE, 
		I_bRedLEDOn:= 		TRUE, 
		I_bRedLEDOff:= 		FALSE, 
		I_diID:= 			I_stInput.diID, 
		I_bOut:= 			I_stInput.bOut, 
		I_sStartZeichen:= 	sStartZeichen, 
		I_sEndZeichen:= 	sEndZeichen,	 
		Q_sConvString=> 	sSendString);
					
	IF GVL_RS485FiFoSend.bSendDoneFiFo[I_FifoID]
	THEN
		sFiFoSend :=	sSendString;
	END_IF
	IF NOT GVL_RS485FiFoSend.bSendDoneFiFo[I_FifoID]
	THEN
		iStepSet := 113;
	END_IF
	
(*============================================================================================*)
113:(* String senden *) (* Warten *)
	IF GVL_RS485FiFoSend.bSendDoneFiFo[I_FifoID]
	THEN
		sFiFoSend := ''; 
		tonStepStartup.IN := TRUE;
		
		IF tonStepStartup.Q
		THEN
			tonStepStartup.IN := FALSE;
			iStepSet := 114;
		END_IF
	END_IF

(*============================================================================================*)
114:(* String senden *)	(* Rote LED Ausschalten *)
	tonStepStartup.IN := FALSE;
	
	fbStringConvR1B6F(
		I_bReset:= 			FALSE, 
		I_bRedLEDOn:= 		FALSE, 
		I_bRedLEDOff:= 		TRUE, 
		I_diID:= 			I_stInput.diID, 
		I_bOut:= 			I_stInput.bOut, 
		I_sStartZeichen:= 	sStartZeichen, 
		I_sEndZeichen:= 	sEndZeichen,	 
		Q_sConvString=> 	sSendString);
			
	IF GVL_RS485FiFoSend.bSendDoneFiFo[I_FifoID]
	THEN
		sFiFoSend :=	sSendString;
	END_IF
	IF NOT GVL_RS485FiFoSend.bSendDoneFiFo[I_FifoID]
	THEN
		iStepSet := 120;
	END_IF
	
(*============================================================================================*)	
120:(* Warten bis nicht Busy *)	
	IF GVL_RS485FiFoSend.bSendDoneFiFo[I_FifoID]
	THEN
		sFiFoSend := ''; 
				
		tonStepStartup.IN := TRUE;
	
		IF tonStepStartup.Q
		THEN
			bStartupDone := TRUE;
			tonStepStartup.IN := FALSE;
			bStartupStart := FALSE;
			iStepSet := 10;	(* Anschließend noch einmal die Eingangs Helligkeit setzen *)
		END_IF
	END_IF	

END_CASE
END_ACTION

ACTION ac01_SetReset:
(*============================================================================================*)
(*	RESET Schrittkette *)
(*============================================================================================*)
tonResetTimeout(
	PT := tResetTimeout);

tonResetDone();

(* Einfaches Setzen der LED Helligkeiten (0-100 Prozent *)
CASE iStepSet OF
(*============================================================================================*)
0:	sStateReset := 'INIT';
	
	IF (bSetExecute
		AND (I_stInput.bReset
		OR bResetAutoStart))
	THEN
		bStartupDone := FALSE;
		bResetDone := FALSE;
		tonResetTimeout.IN := FALSE;
		tonResetDone.IN := FALSE;
		icntResetSend := 0;
		
		(* Ausgänge alle auf 0 setzen *)
		FOR h := 1 TO 16 BY 1 DO
			ibOutMem[h] := FALSE;
			Q_stOutput.bInputs[h] := FALSE;
		END_FOR
		
		bPingOK := FALSE;
		
		iStepSet := iStepSet +1;
	END_IF

(*============================================================================================*)	
1:	sStateReset := 'Sende Reset Befehl';
	bResetBusy := TRUE;
	bErrorReset := FALSE;
	
	fbStringConvR1B6F(
		I_bReset:= 			TRUE, 
		I_bRedLEDOn:= 		FALSE, 
		I_bRedLEDOff:= 		FALSE, 
		I_diID:= 			I_stInput.diID, 
		I_bOut:= 			I_stInput.bOut, 
		I_sStartZeichen:= 	sStartZeichen, 
		I_sEndZeichen:= 	sEndZeichen,	 
		Q_sConvString=> 	sSendString);

	(* Senden an FiFo*)
	IF GVL_RS485FiFoSend.bSendDoneFiFo[I_FifoID]
	THEN
		sFiFoSend :=	sSendString;
	END_IF
	IF NOT GVL_RS485FiFoSend.bSendDoneFiFo[I_FifoID]
	THEN
		iStepSet := iStepSet+1;
	END_IF

(*============================================================================================*)
2:	sStateReset := 'Sende Reset Befehl';

	IF GVL_RS485FiFoSend.bSendDoneFiFo[I_FifoID]
	THEN
		sFiFoSend := ''; 
		
		fbStringConvR1B6F(
			I_bReset :=			FALSE);
		iStepSet := 3;
	END_IF
	
(*============================================================================================*)	
3:	sStateReset := 'Reset durchgeführt, Warte auf Ping';
	tonResetDone.IN := TRUE;
	tonResetDone.PT := tResetReboot;
		
	iState := 0;
	
	IF tonResetDone.Q
	THEN
		tonResetDone.IN := FALSE;
		iStepSet := 4;
	END_IF
	
(*============================================================================================*)	
4:	sStateReset := 'Warte auf Ping vom Gerät';	
	tonResetTimeout.IN := TRUE;
	
	IF bPingOK 
		OR NOT bCheckPing
	THEN
		bErrorReset := FALSE;
		tonResetTimeout.IN := FALSE;
		iStepSet := 5;
	ELSIF
		tonResetTimeout.Q
	THEN
		sStateReset := 'Ping Timeout, keine Kommunikation';
		bErrorReset := TRUE;

		IF I_stInput.bReset
		THEN
			bResetBusy := FALSE;
			iStepSet := 0;
		END_IF
	END_IF

(*============================================================================================*)
5:	sStateReset := 'Startup Aktiv';
	
	tonResetDone.IN := NOT I_stInput.bReset;
	tonResetDone.PT := tResetStartup;

	sFiFoSend := ''; 
	
	IF tonResetDone.Q
	THEN
		fbStringConvR1B6F(
			I_bReset :=			FALSE);
			
		sStateReset := 'Ping erhalten, Reset Erfolgreich';
		bResetAutoStart := FALSE;
		bResetDone := TRUE;
		bResetBusy := FALSE;
		iState := 0;
		iStepSet := 0;
	END_IF
END_CASE
END_ACTION

ACTION ac02_Ping:
(*============================================================================================*)
(* 	Ping Bautsein, Checkt ob die Kommunikation vorhanden ist *)
(*============================================================================================*)
fbRS485ComCheck(
	I_FifoID:=				I_FifoID,
	I_bExecute:= 			bCheckPing
							AND bStartUpCheckPing
							(*AND bReadyToPing*), 
	I_bStart :=				I_bPingStart
							AND bPingFreigabe,
	I_bTasterMode:=			FALSE,
	I_StringReceived:=		I_StringReceived,
	I_tPingIntervall:= 		tPingTimer, 
	I_tPingTimeout:= 		tReceiveTimeout, 
	I_diID:= 				I_stInput.diID, 
	I_sPingSymbol:= 		'.BTN.', 
	I_iInstID:= 			97, 
	I_sStartZeichen:= 		sStartZeichen, 
	I_sEndZeichen:= 		sEndZeichen, 
	I_iMaxPingTry :=		iMaxPingTry,	 
	Q_bComOk=> 				bPingOK, 
	Q_bError=> 				bErrorPing,
	Q_bSendDone=>			(*Q_bPingDone*));
END_ACTION

ACTION ac10_Counter:
(*============================================================================================*)
(* 	Zähler *)
(*============================================================================================*)
FOR j := 1 TO 16 BY 1 DO 
	r_TrigCountBtn[j](
		CLK := I_stInput.bOut[j]);
		
	IF r_TrigCountBtn[j].Q
	THEN
		Q_stCnt.dwCntRelais[j] := Q_stCnt.dwCntRelais[j]+1;
	END_IF
	
END_FOR
END_ACTION

ACTION ac99_Doku:
(*======================================================================================================================================*)
(*	DOKU	*)
(*======================================================================================================================================*)
(* Wichtiger Hinweis:
		-Bei dem 6 Fach Taster ist zu Beachten, dass es nur 4 Externe EA/s gibt also 4 LEDs und 4 Taster, 
		da der ESP 32 Nur 10Es und 10As besitzt.
		- Die 4 Zusätzlichen Ausgänge werden von der Hintergrundbeleuchtung Ausgeschlossen und müssen über den Befehl: SET_MBR einzeln 
			gesetzt werden! *)	
	
(* Verdrahtung:		
	Verdrahtung füR: KL6041
        +-------+
        |       |
        | TxD+ ----+
        |         |----> RS485 A (zum Bus)
        | RxD+ ----+
        |         |
        | TxD− ----+
        |         |----> RS485 B (zum Bus)
        | RxD− ----+
        +-------+	*)
		
(*======================================================================================================================================*)
(* Telegrammbeschreibung *)

(*	Die XML Dateien der verschiedenen Module sind grundsätzlich immer gleich aufgebaut. 
	Je Instanz der verschiedenen Sensoren und Aktoren werden die zu sendenden Befehle bzw. 
	die zu empfangenen Events beschrieben. 
	Alle Telegramme sind ASCII kodiert und sind umgeben mit dem binären Startzeichen 0xFD und dem binären Endezeichen 0xFE.

	Grundaufbauer aller im Folgenden beschriebenen Telegramme:
	
	-Startzeichen immer 0xFD.
	-Punkte dienen als Trennzeichen der verschiedenen Elemente
	-Endezeichen immer 0xFE.
	-Element 1 ist die Geräte-ID, die entsprechend der verwendeten Module angepasst werden muss (hier beispielhaft jeweils 12345)
	-Element 2 ist ein Schlüsselwort für den jeweiligen Funktionstyp (z.b. BTN, LED, DIM, usw)
	-Element 3 ist die InstanzID gemäß XML Templates (also welche Taster oder welcher Dimmer konkret gemeint ist)
	-Element 4 zeigt die jeweilige Aktion zum Funktionstypen (z.b. ON, OFF, STATUS)
	-Anschließend kommen optional diverse Parameter, die mit P1,P2,...P3 bezeichnet werden
	
	Im Folgenden wird nur noch auf die speziellen Telegramdaten eingegangen:
	
	(*------------------------------------------------------------*)
	Taster oder digitaler Eingang (Sensor):
	(*------------------------------------------------------------*)
	Telegram Event:  	
	
	\xFD 12345.BTN.17.STATUS.P1 \xFE
	
		Funktionstyp:		BTN (kurz für Button)
		Instanz-ID:			hier 17 (in XML nachschauen)
		Aktion:				STATUS
		P1:					1, wenn Taste gedrückt bzw. Eingang aktiv
							0, wenn Taste losgelassen bzw. Eingang inaktiv
	
	Telegram Statusabfrage:  	
	
	\xFD 12345.BTN.17.gSTATUS \xFE
	
		Antwort:  			\xFD 12345.BTN.17.rSTATUS.P1 \xFE
		P1:					1, wenn Taste gedrückt bzw. Eingang aktiv
							0, wenn Taste losgelassen bzw. Eingang inaktiv

	(*------------------------------------------------------------*)
	Led (Aktor):
	(*------------------------------------------------------------*)
	Telegram Helligkeit setzen:  	
	
	\xFD 12345.LED.50.ON.P1.P2.P3 \xFE
	
		Funktionstyp:			LED
		Instanz-ID:				hier 50 (in XML nachschauen)
		Aktion:					ON
		P1:						gewünschte Helligkeit 0-100
		P2:						Einschaltdauer in 100stel Sekunden (0 = daueran)
		P3:						Einschaltverzögerung in Sekunden (0 = ohne Verzögerung)
	
	Telegram Mindesthelligkeit:  	
	
	\xFD 12345.LED.50.SET_MBR.P1 \xFE
		
		Aktion:					SET_MBR (Setzt eine Mindesthelligkeit, die auch dann erhalten bleibt, wenn man per OFF ausschaltet)
		P1:						gewünschte Helligkeit 0-100
	
	Telegram Statusabfrage:  	

	\xFD 12345.LED.50.gSTATUS \xFE
	
		Antwort:  				\xFD 12345.LED.50.rSTATUS.P1.P2 \xFE
		P1:						aktuelle Helligkeit 0-100
		P2:						Einschaltdauer in 100stel Sekunden
	
	(*------------------------------------------------------------*)
	Hintergrundbeleuchtung (Aktor):
	(*------------------------------------------------------------*)
	Telegram Minhelligkeit:  
	
	\xFD 12345.LBN.16.SET_MBR.P1 \xFE
	
		Aktion:					SET_MBR ((Setzt eine Mindesthelligkeit, die auch dann erhalten bleibt, wenn man per OFF ausschaltet)
		P1:						gewünschte Helligkeit 0-100
		
	Telegram Statusabfrage:  	

	\xFD 12345.LBN.16.gSTATUS \xFE
	
		Antwort:  				\xFD 12345.LBN.16.rSTATUS.P1 \xFE
		P1:						aktuelle Helligkeit 0-100

	(*------------------------------------------------------------*)
	Temperatursensor (Sensor):
	(*------------------------------------------------------------*)
	Telegram Event:  	
	
	\xFD 12345.TMP.1.STATUS.P1.P2 \xFE
	
		Funktionstyp:			TMP (kurz für Temperatur)
		Instanz-ID:				hier 1 (in XML nachschauen)
		Aktion:					STATUS
		P1:						Temperatur in Grad Vorkommastellen
		P2:						Temperatur in Grad Nachkommastellen
	
	Telegram Statusabfrage:  
	
	\xFD 12345.TMP.1.gSTATUS \xFE
	
		Antwort:  				\xFD 12345.TMP.1.rSTATUS.P1.P2 \xFE
		P1:						Temperatur in Grad Vorkommastellen
		P2:						Temperatur in Grad Nachkommastellen

	(*------------------------------------------------------------*)
	Feuchtesensor (Sensor):
	(*------------------------------------------------------------*)
	Telegram Event:  	

	\xFD 12345.RHD.1.STATUS.P1.P2 \xFE
	
